# B&R Automation Studio project BenchEDM_AS6 (part 3)

#### TC_Recipe.fun - Exported functions and function blocks
```iecst
{REDUND_ERROR} FUNCTION_BLOCK TC_Recipe_Helper (*A helper block for MpRecipe*) (*$GROUP=User,$CAT=User,$GROUPICON=User.png,$CATICON=User.png*)
	VAR_INPUT
		Enable : BOOL;
		Def : Recipe_Definition_typ;
		RemOK : BOOL;
		ErrorReset : BOOL;
		ForceLoad : BOOL;
		ForceSave : BOOL;
		ForceDefaults : BOOL;
	END_VAR
	VAR_OUTPUT
		AutoLoadSuccess : BOOL;
		AutoLoadFailed : BOOL;
		RemLost : BOOL;
		Initialized : BOOL;
		Ready : BOOL;
		Error : BOOL;
	END_VAR
	VAR
		Internal : TC_Recipe_Helper_Internal_typ;
	END_VAR
END_FUNCTION_BLOCK
```

#### TC_Recipe_Helper.st
```iecst
(* A helper block for MpRecipe *)
FUNCTION_BLOCK TC_Recipe_Helper

//Reset in not enabled
	IF NOT Enable THEN
		Internal.State								:= TC_RH_ST_RESET;
	END_IF;

	//Reset Status Flags
	Ready 											:= FALSE;
	Error											:= FALSE;
	AutoLoadSuccess									:= FALSE;
	AutoLoadFailed									:= FALSE;
	RemLost											:= FALSE;

	//Main Case
	CASE Internal.State OF
		TC_RH_ST_RESET:
			Initialized								:= FALSE;
			Internal.ErrorReset 					:= FALSE;
			Internal.MpRecipeXml_0.Load				:= FALSE;
			Internal.MpRecipeXml_0.Save				:= FALSE;
			Internal.State							:= TC_RH_ST_VALIDATE_INPUTS;
		TC_RH_ST_VALIDATE_INPUTS:
			IF Def.pVar = 0 OR Def.SizeVar = 0 OR Def.DeviceName = '' OR Def.FileName = '' OR Def.VarName = '' THEN
				Internal.State						:= TC_RH_ST_ERROR;
			ELSE
				Internal.State						:= TC_RH_ST_REG_PAR_W;
			END_IF;
		TC_RH_ST_REG_PAR_W:
			Internal.CTON_Timeout.IN				:= TRUE;
			Internal.CTON_Timeout.PT				:= T#2s;
			IF Internal.MpRecipeRegPar_0.Error THEN
				Internal.State						:= TC_RH_ST_ERROR;
			ELSIF Internal.CTON_Timeout.Q THEN
				Internal.State						:= TC_RH_ST_ERROR;
			ELSIF Internal.MpRecipeRegPar_0.Active THEN
				IF RemOK THEN
					Internal.State					:= TC_RH_ST_READY;
				ELSE
					RemLost							:= TRUE;
					Internal.MpRecipeXml_0.Load		:= TRUE;
					Internal.State					:= TC_RH_ST_AUTO_LOAD_W;
				END_IF;
			END_IF;
		TC_RH_ST_READY:
			IF ForceLoad THEN
				Internal.MpRecipeXml_0.Load			:= TRUE;
				Internal.State						:= TC_RH_ST_LOAD_W;
			ELSIF ForceDefaults THEN
				IF Def.pDefaultVar <> 0 THEN
					brsmemcpy(Def.pVar,Def.pDefaultVar,Def.SizeVar);
				ELSE
					brsmemset(Def.pVar,0,Def.SizeVar);
				END_IF;
				Internal.MpRecipeXml_0.Save			:= TRUE;
				Internal.State						:= TC_RH_ST_SAVE_W;
			ELSIF ForceSave THEN
				Internal.MpRecipeXml_0.Save			:= TRUE;
				Internal.State						:= TC_RH_ST_SAVE_W;
			ELSIF Def.pCmpVar <> 0 THEN //AutoSave Enabled
				IF brsmemcmp(Def.pCmpVar,Def.pVar,Def.SizeVar) <> 0 THEN //AutoSave On Change
					brsmemcpy(Def.pCmpVar,Def.pVar,Def.SizeVar);
					Internal.MpRecipeXml_0.Save		:= TRUE;
					Internal.State					:= TC_RH_ST_SAVE_W;
				ELSE
					Ready 							:= TRUE;
					Initialized						:= TRUE;
				END_IF;
			ELSE
				Initialized							:= TRUE;
				Ready 								:= TRUE;
			END_IF;
		TC_RH_ST_LOAD_W:
			Internal.CTON_Timeout.IN				:= TRUE;
			Internal.CTON_Timeout.PT				:= T#2s;
			IF (NOT Internal.MpRecipeXml_0.CommandBusy AND Internal.MpRecipeXml_0.Error) OR Internal.CTON_Timeout.Q THEN
				Internal.MpRecipeXml_0.Load			:= FALSE;
				Internal.State						:= TC_RH_ST_ERROR;
			ELSIF (NOT Internal.MpRecipeXml_0.CommandBusy AND Internal.MpRecipeXml_0.CommandDone AND NOT Internal.MpRecipeXml_0.Error) THEN
				Internal.MpRecipeXml_0.Load			:= FALSE;
				Internal.State						:= TC_RH_ST_READY;
			END_IF;
		TC_RH_ST_SAVE_W:
			Internal.CTON_Timeout.IN				:= TRUE;
			Internal.CTON_Timeout.PT				:= T#2s;
			IF (NOT Internal.MpRecipeXml_0.CommandBusy AND Internal.MpRecipeXml_0.Error) OR Internal.CTON_Timeout.Q THEN
				Internal.MpRecipeXml_0.Save			:= FALSE;
				Internal.State						:= TC_RH_ST_ERROR;
			ELSIF (NOT Internal.MpRecipeXml_0.CommandBusy AND Internal.MpRecipeXml_0.CommandDone AND NOT Internal.MpRecipeXml_0.Error) THEN
				Internal.MpRecipeXml_0.Save			:= FALSE;
				Internal.State						:= TC_RH_ST_READY;
			END_IF;
		TC_RH_ST_AUTO_LOAD_W:
			Internal.CTON_Timeout.IN				:= TRUE;
			Internal.CTON_Timeout.PT				:= T#2s;
			IF (NOT Internal.MpRecipeXml_0.CommandBusy AND Internal.MpRecipeXml_0.Error) OR Internal.CTON_Timeout.Q THEN
				AutoLoadFailed						:= TRUE;
				IF Def.pDefaultVar <> 0 THEN
					brsmemcpy(Def.pVar,Def.pDefaultVar,Def.SizeVar);
				ELSE
					brsmemset(Def.pVar,0,Def.SizeVar);
				END_IF;
				Internal.MpRecipeXml_0.Load			:= FALSE;
				Internal.State						:= TC_RH_ST_AUTO_RESET_D;
			ELSIF (NOT Internal.MpRecipeXml_0.CommandBusy AND Internal.MpRecipeXml_0.CommandDone AND NOT Internal.MpRecipeXml_0.Error) THEN
				AutoLoadSuccess						:= TRUE;
				Internal.MpRecipeXml_0.Load			:= FALSE;
				Internal.State						:= TC_RH_ST_READY;
			END_IF;
		TC_RH_ST_AUTO_RESET_D:
			Internal.State							:= TC_RH_ST_AUTO_RESET_C;
		TC_RH_ST_AUTO_RESET_C:
			Internal.ErrorReset						:= TRUE;
			Internal.State							:= TC_RH_ST_AUTO_RESET_W;
		TC_RH_ST_AUTO_RESET_W:
			Internal.CTON_Timeout.IN				:= TRUE;
			Internal.CTON_Timeout.PT				:= T#2s;
			IF Internal.CTON_Timeout.Q THEN
				Internal.ErrorReset					:= FALSE;
				Internal.State						:= TC_RH_ST_ERROR;
			ELSIF NOT Internal.MpRecipeXml_0.Error THEN
				Internal.ErrorReset					:= FALSE;
				Internal.MpRecipeXml_0.Save			:= TRUE;
				Internal.State						:= TC_RH_ST_AUTO_SAVE_W;
			END_IF;
		TC_RH_ST_AUTO_SAVE_W:
			Internal.CTON_Timeout.IN				:= TRUE;
			Internal.CTON_Timeout.PT				:= T#2s;
			IF (NOT Internal.MpRecipeXml_0.CommandBusy AND Internal.MpRecipeXml_0.Error) OR Internal.CTON_Timeout.Q THEN
				Internal.MpRecipeXml_0.Save			:= FALSE;
				Internal.State						:= TC_RH_ST_ERROR;
			ELSIF (NOT Internal.MpRecipeXml_0.CommandBusy AND Internal.MpRecipeXml_0.CommandDone AND NOT Internal.MpRecipeXml_0.Error) THEN
				Internal.MpRecipeXml_0.Save			:= FALSE;
				Internal.State						:= TC_RH_ST_READY;
			END_IF;
		TC_RH_ST_ERROR:
			Error									:= TRUE;
			IF ErrorReset THEN
				Internal.State						:= TC_RH_ST_RESET;
			END_IF;
	END_CASE;

	//Reset Commands
	ForceDefaults 									:= FALSE;
	ForceLoad 										:= FALSE;
	ForceSave 										:= FALSE;

	//Reset Timeout On State Change
	IF Internal.LastState <> Internal.State OR Internal.State = TC_RH_ST_RESET THEN
		Internal.LastState 							:= Internal.State;
		Internal.CTON_Timeout.IN					:= FALSE;
	END_IF;

	//FB Calls
	Internal.CTON_Timeout();
	Internal.MpRecipeRegPar_0(MpLink := ADR(Def.MpLink), Enable := Enable, ErrorReset := (ErrorReset OR Internal.ErrorReset), PVName := ADR(Def.VarName), Category := ADR(Def.VarName));
	Internal.MpRecipeXml_0(MpLink := ADR(Def.MpLink), Enable := Enable, ErrorReset := (ErrorReset OR Internal.ErrorReset), DeviceName := ADR(Def.DeviceName), FileName := ADR(Def.FileName), Category := ADR(Def.VarName));

END_FUNCTION_BLOCK
```

### Library Logical/Libraries/TC_Sim (IEC)
Depends on: MTTypes, MTBasics, MTFilter

#### Types.typ - Exported data types
```iecst
TYPE
	TC_Sim_Actuator_TF_Internal_typ : 	STRUCT
		Active : BOOL;
		OldDampingRatio : REAL;
		OldNaturalFreq : REAL;
		OldFullStrokeValue : REAL;
		MTBasicsTransferFcn_0 : MTBasicsTransferFcn;
	END_STRUCT;
	TC_Sim_Actuator_Lin_Internal_typ : 	STRUCT
		Active : BOOL;
		OldTimePos : REAL;
		OldTimeNeg : REAL;
		MTBasicsLimiter_0 : MTBasicsLimiter;
	END_STRUCT;
END_TYPE
```

#### TC_Sim.fun - Exported functions and function blocks
```iecst
{REDUND_ERROR} FUNCTION_BLOCK TC_Sim_Actuator_Lin (* *) (*$GROUP=User,$CAT=User,$GROUPICON=User.png,$CATICON=User.png*)
	VAR_INPUT
		Enable : BOOL;
		Actuate : BOOL;
		FullStrokeValue : REAL;
		FeedbackTol : REAL;
		TimeNeg : REAL;
		TimePos : REAL;
	END_VAR
	VAR_OUTPUT
		Position : REAL;
		AtFalsePosition : BOOL;
		AtTruePosition : BOOL;
		Error : BOOL;
	END_VAR
	VAR
		Internal : TC_Sim_Actuator_Lin_Internal_typ;
	END_VAR
END_FUNCTION_BLOCK

{REDUND_ERROR} FUNCTION_BLOCK TC_Sim_Actuator_TF (* *) (*$GROUP=User,$CAT=User,$GROUPICON=User.png,$CATICON=User.png*)
	VAR_INPUT
		Enable : BOOL;
		Actuate : BOOL;
		ClampValueToEnds : BOOL;
		FullStrokeValue : REAL;
		FeedbackTol : REAL;
		NaturalFreq : REAL;
		DampingRatio : REAL;
	END_VAR
	VAR_OUTPUT
		Position : REAL;
		AtFalsePosition : BOOL;
		AtTruePosition : BOOL;
		Error : BOOL;
	END_VAR
	VAR
		Internal : TC_Sim_Actuator_TF_Internal_typ;
	END_VAR
END_FUNCTION_BLOCK
```

#### TC_Sim_Actuator_TF.st
```iecst
FUNCTION_BLOCK TC_Sim_Actuator_TF

	IF Enable THEN
		IF NOT Internal.Active OR (Internal.Active AND (Internal.OldNaturalFreq <> NaturalFreq OR Internal.OldDampingRatio <> DampingRatio OR Internal.OldFullStrokeValue <> FullStrokeValue)) THEN
			Internal.MTBasicsTransferFcn_0.Numerator[0] 	:= FullStrokeValue*NaturalFreq**2;
			Internal.MTBasicsTransferFcn_0.Denominator[0] 	:= NaturalFreq**2;
			Internal.MTBasicsTransferFcn_0.Denominator[1] 	:= 2*DampingRatio*NaturalFreq;
			Internal.MTBasicsTransferFcn_0.Denominator[2] 	:= 1;
			Internal.OldNaturalFreq							:= NaturalFreq;
			Internal.OldDampingRatio						:= DampingRatio;
			Internal.OldFullStrokeValue						:= FullStrokeValue;
			IF Internal.Active THEN
				Internal.MTBasicsTransferFcn_0.Update		:= TRUE;
			END_IF;
			Internal.Active 								:= TRUE;
		END_IF;

		IF Actuate THEN
			Internal.MTBasicsTransferFcn_0.In				:= 1.0;
		ELSE
			Internal.MTBasicsTransferFcn_0.In				:= 0.0;
		END_IF;

		Position 											:= Internal.MTBasicsTransferFcn_0.Out;
		IF ClampValueToEnds THEN
			IF Internal.MTBasicsTransferFcn_0.Out > FullStrokeValue THEN
				Position 									:= FullStrokeValue;
			ELSIF Internal.MTBasicsTransferFcn_0.Out < 0 THEN
				Position 									:= 0.0;
			END_IF;
		END_IF;

		AtFalsePosition										:= ABS(Position) <= FeedbackTol;
		AtTruePosition										:= ABS(Position-FullStrokeValue) <= FeedbackTol;
		Internal.MTBasicsTransferFcn_0.Enable				:= TRUE;
	ELSE
		Position 											:= 0.0;
		AtFalsePosition 									:= FALSE;
		AtTruePosition 										:= FALSE;
		Internal.Active 									:= FALSE;
		Internal.MTBasicsTransferFcn_0.Enable				:= FALSE;
		Internal.MTBasicsTransferFcn_0.In					:= 0.0;
		Internal.OldNaturalFreq								:= 0.0;
		Internal.OldDampingRatio							:= 0.0;
		Internal.OldFullStrokeValue							:= 0.0;
	END_IF;

	Internal.MTBasicsTransferFcn_0();
	Internal.MTBasicsTransferFcn_0.Update 					:= FALSE;
	Error 													:= Internal.MTBasicsTransferFcn_0.Error;

END_FUNCTION_BLOCK
```

#### TC_Sim_Actuator_Lin.st
```iecst
FUNCTION_BLOCK TC_Sim_Actuator_Lin

	IF Enable THEN
		IF NOT Internal.Active OR (Internal.Active AND (Internal.OldTimeNeg <> TimeNeg OR Internal.OldTimePos <> TimePos)) THEN
			IF TimeNeg <= 0 THEN
				Internal.MTBasicsLimiter_0.MaxNegSlewRate	:= 0;
			ELSE
				Internal.MTBasicsLimiter_0.MaxNegSlewRate	:= 1.0/TimeNeg;
			END_IF;
			IF TimePos <= 0 THEN
				Internal.MTBasicsLimiter_0.MaxPosSlewRate	:= 0;
			ELSE
				Internal.MTBasicsLimiter_0.MaxPosSlewRate	:= 1.0/TimePos;
			END_IF;
			Internal.OldTimeNeg 							:= TimeNeg;
			Internal.OldTimePos 							:= TimePos;
			IF Internal.Active THEN
				Internal.MTBasicsLimiter_0.Update			:= TRUE;
			END_IF;
			Internal.Active 								:= TRUE;
		END_IF;

		IF Actuate THEN
			Internal.MTBasicsLimiter_0.In					:= 1.0;
		ELSE
			Internal.MTBasicsLimiter_0.In					:= 0.0;
		END_IF;

		Position 											:= Internal.MTBasicsLimiter_0.Out*FullStrokeValue;

		AtFalsePosition										:= ABS(Position) <= FeedbackTol;
		AtTruePosition										:= ABS(Position-FullStrokeValue) <= FeedbackTol;
		Internal.MTBasicsLimiter_0.Enable					:= TRUE;
	ELSE
		Position 											:= 0.0;
		AtFalsePosition 									:= FALSE;
		AtTruePosition 										:= FALSE;
		Internal.Active 									:= FALSE;
		Internal.MTBasicsLimiter_0.Enable					:= FALSE;
		Internal.MTBasicsLimiter_0.In						:= 0.0;
		Internal.OldTimeNeg									:= 0.0;
		Internal.OldTimePos									:= 0.0;
	END_IF;

	Internal.MTBasicsLimiter_0();
	Internal.MTBasicsLimiter_0.Update 						:= FALSE;
	Error 													:= Internal.MTBasicsLimiter_0.Error;

END_FUNCTION_BLOCK
```

### Library Logical/Libraries/TC_AlarmX (IEC)
Depends on: AsBrStr, TC_General, TC_Str, MpAlarmX, MpBase

#### Types.typ - Exported data types
```iecst
TYPE
	TC_AlarmX_Helper_Internal_typ : 	STRUCT
		Active : BOOL;
		AddText : STRING[1000];
		ArEventLogGetIdent_0 : ArEventLogGetIdent;
		ArEventLogWrite_0 : ArEventLogWrite;
	END_STRUCT;
	TC_ALARMX_ACTION_ENUM :
		(
		TC_ALARMX_ACTION_NONE,
		TC_ALARMX_ACTION_SET,
		TC_ALARMX_ACTION_SET_NO_LOG,
		TC_ALARMX_ACTION_ACK,
		TC_ALARMX_ACTION_ACK_NO_LOG,
		TC_ALARMX_ACTION_LOG_ONLY
		);
	TC_ALARMX_CORE_STATE_ENUM :
		(
		TC_ALARMX_CORE_RESET,
		TC_ALARMX_CORE_IDLE,
		TC_ALARMX_CORE_SET_C,
		TC_ALARMX_CORE_SET_W
		);
	TC_AlarmX_Core_Internal_typ : 	STRUCT
		state : TC_ALARMX_CORE_STATE_ENUM;
		currentAlarm : TC_AlarmX_Core_Buffer_typ;
		tDelay : CTON;
		i : INT;
	END_STRUCT;
	TC_AlarmX_Core_Buffer_typ : 	STRUCT
		name : STRING[MAX_ALARM_NAME_LEN];
		addText : ARRAY[0..TC_ALARMX_MAX_ADD_DATA_IDX]OF STRING[MAX_ALARM_ADD_DATA];
		allowMultiple : BOOL;
	END_STRUCT;
	TC_AlarmX_AlarmExtraData_typ : 	STRUCT
		AddData : ARRAY[0..TC_ALARMX_MAX_ADD_DATA_IDX]OF STRING[MAX_ALARM_ADD_DATA];
	END_STRUCT;
	TC_AlarmX_CfgMod_Internal_typ : 	STRUCT
		AlarmName : STRING[MAX_ALARM_NAME_LEN];
		i : USINT;
		CTON_Timeout : CTON;
	END_STRUCT;
	TC_AlarmX_BufferInfo_typ : 	STRUCT
		Address : UDINT;
		Size : UDINT;
	END_STRUCT;
	TC_Module_Alarm_Info_typ : 	STRUCT
		ErrorInfo : USINT;
		IgnoreInfo : USINT;
	END_STRUCT;
END_TYPE
```

#### Constants.var - Exported constants
```iecst
VAR CONSTANT
	TC_MODULE_MAX_ALARM : USINT := 6;
	MAX_ALARM_ADD_DATA : UDINT := 255; (*Maximum Length of the extra alarm text*)
	MAX_ALARM_NAME_LEN : UDINT := 255; (*Maximum Length of the alarm name*)
	TC_ALARMX_BUFFER_IDX : UDINT := 255; (*Length of alarm buffer*)
	TC_ALARMX_MAX_ADD_DATA_IDX : USINT := 3;
END_VAR
```

#### TC_AlarmX.fun - Exported functions and function blocks
```iecst
{REDUND_ERROR} FUNCTION TC_AlarmX_Helper : DINT (*Helper Function for Setting and Acknowledging Alarms with User Logger support.*) (*$GROUP=User,$CAT=User,$GROUPICON=User.png,$CATICON=User.png*)
	VAR_INPUT
		MpLink : MpComIdentType;
		AlarmName : STRING[255];
		AlarmAction : TC_ALARMX_ACTION_ENUM;
		LogEventAddText : STRING[255];
		AllowMultiple : BOOL;
	END_VAR
	VAR
		Internal : TC_AlarmX_Helper_Internal_typ;
	END_VAR
END_FUNCTION

{REDUND_ERROR} FUNCTION_BLOCK TC_AlarmXCore (*TODO: Add your comment here*) (*$GROUP=User,$CAT=User,$GROUPICON=User.png,$CATICON=User.png*)
	VAR_INPUT
		enable : BOOL;
		MpLink : MpComIdentType;
		pBuffer : UDINT;
		pOutputData : REFERENCE TO TC_AlarmX_AlarmExtraData_typ;
		delayTime : TIME;
	END_VAR
	VAR
		internal : TC_AlarmX_Core_Internal_typ;
	END_VAR
END_FUNCTION_BLOCK
```

#### TC_AlarmX_Helper.st
```iecst
(* Helper Function for Setting and Acknowledging Alarms with User Logger support. *)
FUNCTION TC_AlarmX_Helper
	TC_AlarmX_Helper 					:= -1;
	brsmemset(ADR(Internal),0,SIZEOF(Internal));
	Internal.ArEventLogGetIdent_0(Execute := FALSE);
	Internal.ArEventLogGetIdent_0(Execute := TRUE, Name := '$$arlogusr');
	Internal.AddText 					:= AlarmName;
	Internal.Active						:= NOT MpAlarmXCheckState(MpLink,AlarmName,mpALARMX_STATE_NONE);

	CASE AlarmAction OF
		TC_ALARMX_ACTION_NONE:
			TC_AlarmX_Helper 			:= 0;
		TC_ALARMX_ACTION_SET:
			TC_AlarmX_Helper 			:= 0;
			IF NOT Internal.Active OR AllowMultiple THEN
				MpAlarmXSet(MpLink,AlarmName);
				brsmemset(ADR(Internal.AddText),0,SIZEOF(Internal.AddText));
				Internal.AddText 	:= AlarmName;
				TC_brsstrcat(ADR(Internal.AddText),ADR(' - Set'),SIZEOF(Internal.AddText));
				IF LogEventAddText <> '' THEN
					TC_brsstrcat(ADR(Internal.AddText),ADR(' - Info: '),SIZEOF(Internal.AddText));
					TC_brsstrcat(ADR(Internal.AddText),ADR(LogEventAddText),SIZEOF(Internal.AddText));
				END_IF;
				Internal.ArEventLogWrite_0(Execute := FALSE);
				Internal.ArEventLogWrite_0(Execute := TRUE, Ident := Internal.ArEventLogGetIdent_0.Ident, EventID := -536870912, OriginRecordID := 0, ObjectID := 'TC_AlarmX_Helper', AddDataSize := brsstrlen(ADR(Internal.AddText)), AddDataFormat := 1, AddData := ADR(Internal.AddText), TimeStamp := 0);
			END_IF;
		TC_ALARMX_ACTION_SET_NO_LOG:
			TC_AlarmX_Helper 			:= 0;
			IF NOT Internal.Active OR AllowMultiple THEN
				MpAlarmXSet(MpLink,AlarmName);
				brsmemset(ADR(Internal.AddText),0,SIZEOF(Internal.AddText));
			END_IF;
		TC_ALARMX_ACTION_ACK:
			TC_AlarmX_Helper 			:= 0;
			IF Internal.Active THEN
				MpAlarmXAcknowledge(MpLink,AlarmName);
				brsmemset(ADR(Internal.AddText),0,SIZEOF(Internal.AddText));
				Internal.AddText 	:= AlarmName;
				TC_brsstrcat(ADR(Internal.AddText),ADR(' - Ack'),SIZEOF(Internal.AddText));
				IF LogEventAddText <> '' THEN
					TC_brsstrcat(ADR(Internal.AddText),ADR(' - Info: '),SIZEOF(Internal.AddText));
					TC_brsstrcat(ADR(Internal.AddText),ADR(LogEventAddText),SIZEOF(Internal.AddText));
				END_IF;
				Internal.ArEventLogWrite_0(Execute := FALSE);
				Internal.ArEventLogWrite_0(Execute := TRUE, Ident := Internal.ArEventLogGetIdent_0.Ident, EventID := -536870912, OriginRecordID := 0, ObjectID := 'TC_AlarmX_Helper', AddDataSize := brsstrlen(ADR(Internal.AddText)), AddDataFormat := 1, AddData := ADR(Internal.AddText), TimeStamp := 0);
			END_IF;
		TC_ALARMX_ACTION_ACK_NO_LOG:
			TC_AlarmX_Helper 			:= 0;
			IF Internal.Active THEN
				MpAlarmXAcknowledge(MpLink,AlarmName);
			END_IF;
		TC_ALARMX_ACTION_LOG_ONLY:
			TC_AlarmX_Helper 			:= 0;
			brsmemset(ADR(Internal.AddText),0,SIZEOF(Internal.AddText));
			IF LogEventAddText <> '' THEN
				TC_brsstrcat(ADR(Internal.AddText),ADR('Info: '),SIZEOF(Internal.AddText));
				TC_brsstrcat(ADR(Internal.AddText),ADR(LogEventAddText),SIZEOF(Internal.AddText));
				Internal.ArEventLogWrite_0(Execute := FALSE);
				Internal.ArEventLogWrite_0(Execute := TRUE, Ident := Internal.ArEventLogGetIdent_0.Ident, EventID := -536870912, OriginRecordID := 0, ObjectID := 'TC_AlarmX_Helper', AddDataSize := brsstrlen(ADR(Internal.AddText)), AddDataFormat := 1, AddData := ADR(Internal.AddText), TimeStamp := 0);
			END_IF;
	END_CASE;

END_FUNCTION
```

#### TC_AlarmXCore.st
```iecst
(* Alarm Core to handle setting multiple alarms in one cycle with different texts *)
FUNCTION_BLOCK TC_AlarmXCore

	IF enable = FALSE THEN
		internal.state := TC_ALARMX_CORE_RESET;
	END_IF

	CASE internal.state OF

		TC_ALARMX_CORE_RESET:

			brsmemset(ADR(internal.currentAlarm), 0, SIZEOF(internal.currentAlarm));
			internal.state := TC_ALARMX_CORE_IDLE;

		TC_ALARMX_CORE_IDLE:

			IF TC_Array_PeekBtm(pBuffer, SIZEOF(internal.currentAlarm) * TC_ALARMX_BUFFER_IDX, ADR(internal.currentAlarm), SIZEOF(internal.currentAlarm)) > 0 THEN
				TC_Array_Dequeue(pBuffer, SIZEOF(internal.currentAlarm) * TC_ALARMX_BUFFER_IDX, ADR(internal.currentAlarm), SIZEOF(internal.currentAlarm));
				internal.state := TC_ALARMX_CORE_SET_C;
			END_IF

		TC_ALARMX_CORE_SET_C:

			FOR internal.i := 0 TO TC_ALARMX_MAX_ADD_DATA_IDX DO
				pOutputData.AddData[internal.i]	:= internal.currentAlarm.addText[internal.i];
			END_FOR
			TC_AlarmX_Helper(MpLink, internal.currentAlarm.name, TC_ALARMX_ACTION_SET, '', internal.currentAlarm.allowMultiple);

			internal.state := TC_ALARMX_CORE_SET_W;

		TC_ALARMX_CORE_SET_W:

			internal.tDelay.IN	:= TRUE;
			internal.tDelay.PT	:= delayTime;

			IF internal.tDelay.Q THEN
				internal.tDelay.IN	:= FALSE;
				internal.state 		:= TC_ALARMX_CORE_IDLE;
			END_IF

	END_CASE

	internal.tDelay();

END_FUNCTION_BLOCK
```

### Library Logical/Libraries/TC_Str (IEC)

#### Types.typ - Exported data types
```iecst
TYPE
	TC_brsstrcat_Internal_typ : 	STRUCT
		SrcSize : UDINT;
		DestSize : UDINT;
	END_STRUCT;
	TC_Find_Extract_Internal_typ : 	STRUCT
		i : UDINT;
		sB : UDINT;
		sSL : UDINT;
		sSR : UDINT;
		Len : UDINT;
		Pos : UDINT;
		P1 : DINT;
		P2 : DINT;
	END_STRUCT;
	TC_Find_S_Internal_typ : 	STRUCT
		i : UDINT;
		sB : UDINT;
		sS : UDINT;
	END_STRUCT;
	TC_Find_R_Internal_typ : 	STRUCT
		i : UDINT;
		sB : UDINT;
		sS : UDINT;
	END_STRUCT;
	TC_Find_L_Internal_typ : 	STRUCT
		i : UDINT;
		sB : UDINT;
		sS : UDINT;
	END_STRUCT;
END_TYPE
```

#### TC_Str.fun - Exported functions and function blocks
```iecst
FUNCTION TC_brsstrcat : BOOL
	VAR_INPUT
		pDest : UDINT;
		pSrc : UDINT;
		DestSize : UDINT;
	END_VAR
	VAR
		Internal : TC_brsstrcat_Internal_typ;
	END_VAR
END_FUNCTION

{REDUND_ERROR} FUNCTION TC_Find_L : DINT (*Returns index of substring. Negative values are Errors.*) (*$GROUP=User,$CAT=User,$GROUPICON=User.png,$CATICON=User.png*)
	VAR_INPUT
		pBuffer : UDINT;
		pSearch : UDINT;
	END_VAR
	VAR
		Internal : TC_Find_L_Internal_typ;
	END_VAR
END_FUNCTION

{REDUND_ERROR} FUNCTION TC_Find_R : DINT (*Returns right index of substring. Negative values are Errors.*) (*$GROUP=User,$CAT=User,$GROUPICON=User.png,$CATICON=User.png*)
	VAR_INPUT
		pBuffer : UDINT;
		pSearch : UDINT;
	END_VAR
	VAR
		Internal : TC_Find_R_Internal_typ;
	END_VAR
END_FUNCTION

{REDUND_ERROR} FUNCTION TC_Find_S : DINT (*Returns right index of substring. Negative values are Errors.*) (*$GROUP=User,$CAT=User,$GROUPICON=User.png,$CATICON=User.png*)
	VAR_INPUT
		pBuffer : UDINT;
		pSearch : UDINT;
	END_VAR
	VAR
		Internal : TC_Find_S_Internal_typ;
	END_VAR
END_FUNCTION

{REDUND_ERROR} FUNCTION TC_Find_Extract : DINT (*Returns end position for next search. Negative values are Errors.*) (*$GROUP=User,$CAT=User,$GROUPICON=User.png,$CATICON=User.png*)
	VAR_INPUT
		pBuffer : UDINT;
		pSearchL : UDINT;
		pSearchR : UDINT;
		pExtractADR : UDINT;
		pExtractSIZEOF : UDINT;
	END_VAR
	VAR
		Internal : TC_Find_Extract_Internal_typ;
	END_VAR
END_FUNCTION
```

#### TC_brsstrcat.st
```iecst
(* Checks the memory area before concatenating to prevent overrun. Returns false and doesnt concat if overrun is detected *)
FUNCTION TC_brsstrcat
	TC_brsstrcat 						:= TRUE;
	IF pSrc = 0 OR pDest = 0 OR DestSize = 0 THEN
		TC_brsstrcat 					:= FALSE;
	ELSE
		TC_brsstrcat					:= TRUE;
		brsmemset(ADR(Internal),0,SIZEOF(Internal));
		Internal.SrcSize := brsstrlen(pSrc);
		Internal.DestSize := brsstrlen(pDest);
		IF (Internal.SrcSize+Internal.DestSize) <= DestSize-1 THEN
			brsstrcat(pDest,pSrc);
		ELSE
			TC_brsstrcat				:= FALSE;
		END_IF;
	END_IF;
END_FUNCTION
```

#### TC_Find_S.st
```iecst
(* Returns Right index of substring, substring only returns result if found at START of buffer. Negative values are Errors. *)
FUNCTION TC_Find_S
	IF pBuffer = 0 OR pSearch = 0 THEN
		TC_Find_S	 						:= -2;
	ELSE
		Internal.sB							:= brsstrlen(pBuffer);
		Internal.sS							:= brsstrlen(pSearch);
		IF Internal.sB = 0 OR Internal.sB < Internal.sS THEN
		TC_Find_S	 						:= -3;
		END_IF;
	END_IF;
	IF TC_Find_S = 0 THEN
		TC_Find_S							:= -1;
		IF Internal.sS = 0 THEN
			TC_Find_S 						:= 0;
			RETURN;
		ELSE
			FOR Internal.i := 0 TO Internal.sB-Internal.sS DO
				IF brsmemcmp(pBuffer+Internal.i,pSearch,Internal.sS) = 0 THEN
					TC_Find_S 				:= Internal.i+Internal.sS;
					RETURN;
				ELSE
					RETURN;
				END_IF;
			END_FOR;
		END_IF;
	END_IF;
END_FUNCTION
```

#### TC_Find_L.st
```iecst
(* Returns Left index of substring. Negative values are Errors. *)
FUNCTION TC_Find_L
	IF pBuffer = 0 OR pSearch = 0 THEN
		TC_Find_L	 						:= -2;
	ELSE
		Internal.sB							:= brsstrlen(pBuffer);
		Internal.sS							:= brsstrlen(pSearch);
		IF Internal.sB = 0 OR Internal.sB < Internal.sS THEN
			TC_Find_L	 					:= -3;
		END_IF;
	END_IF;
	IF TC_Find_L = 0 THEN
		TC_Find_L							:= -1;
		IF Internal.sS = 0 THEN
			TC_Find_L 						:= 0;
			RETURN;
		ELSE
			FOR Internal.i := 0 TO Internal.sB-Internal.sS DO
				IF brsmemcmp(pBuffer+Internal.i,pSearch,Internal.sS) = 0 THEN
					TC_Find_L 				:= Internal.i;
					RETURN;
				END_IF;
			END_FOR;
		END_IF;
	END_IF;
END_FUNCTION
```

#### TC_Find_R.st
```iecst
(* Returns Right index of substring. Negative values are Errors. *)
FUNCTION TC_Find_R
	IF pBuffer = 0 OR pSearch = 0 THEN
		TC_Find_R	 						:= -2;
	ELSE
		Internal.sB							:= brsstrlen(pBuffer);
		Internal.sS							:= brsstrlen(pSearch);
		IF Internal.sB = 0 OR Internal.sB < Internal.sS THEN
		TC_Find_R	 						:= -3;
		END_IF;
	END_IF;
	IF TC_Find_R = 0 THEN
		TC_Find_R							:= -1;
		IF Internal.sS = 0 THEN
			TC_Find_R 						:= 0;
			RETURN;
		ELSE
			FOR Internal.i := 0 TO Internal.sB-Internal.sS DO
				IF brsmemcmp(pBuffer+Internal.i,pSearch,Internal.sS) = 0 THEN
					TC_Find_R 				:= Internal.i+Internal.sS;
					RETURN;
				END_IF;
			END_FOR;
		END_IF;
	END_IF;
END_FUNCTION
```

#### TC_Find_Extract.st
```iecst
(* Negative values are Errors. *)
FUNCTION TC_Find_Extract
	IF pBuffer = 0 OR pSearchL = 0 OR pSearchR = 0 OR pExtractADR = 0 OR pExtractSIZEOF = 0 THEN
		TC_Find_Extract 						:= -2;
	ELSE
		Internal.sB								:= brsstrlen(pBuffer);
		Internal.sSL							:= brsstrlen(pSearchL);
		Internal.sSR							:= brsstrlen(pSearchR);
		IF Internal.sB = 0 OR Internal.sB < (Internal.sSL + Internal.sSR + 1) THEN
			TC_Find_Extract 					:= -3;
		END_IF;
	END_IF;
	IF TC_Find_Extract = 0 THEN
		TC_Find_Extract							:= -1;
		Internal.P1 							:= TC_Find_R(pBuffer,pSearchL);
		IF Internal.P1 >= 0 THEN
			Internal.P2 						:= TC_Find_L(pBuffer+Internal.P1,pSearchR);
			IF Internal.P2 >= 0 THEN
				Internal.Pos 					:= Internal.P1 + pBuffer;
				Internal.Len 					:= DINT_TO_UDINT(Internal.P2);
				brsmemcpy(pExtractADR,ADR(Internal.Pos),4);
				brsmemcpy(pExtractSIZEOF,ADR(Internal.Len),4);
				TC_Find_Extract					:= Internal.P1+Internal.P2+Internal.sSR;
			END_IF;
		END_IF;
	END_IF;
END_FUNCTION
```

### Library Logical/Libraries/TC_JSON (IEC)
Depends on: TC_Str, AsBrStr, sys_lib

#### TC_JSON.fun - Exported functions and function blocks
```iecst
{REDUND_ERROR} FUNCTION_BLOCK TC_JSON_PairsToJSON (*FB parses a JSON string into a flat array of Name and Value Pairs*) (*$GROUP=User,$CAT=User,$GROUPICON=User.png,$CATICON=User.png*)
	VAR_INPUT
		Enable : BOOL;
		pBuffer : UDINT; (*Pointer to Buffer*)
		BufferSIZEOF : UDINT; (*Buffer SIZEOF*)
		pPairs : UDINT; (*Pointer to Array defined as HA_JSON_Parse_Pair_typ[0..MAX_JSON_PARSE_PAIR_IDX]*)
	END_VAR
	VAR_OUTPUT
		Done : BOOL;
		Error : BOOL;
	END_VAR
	VAR
		Internal : TC_JSON_PairsToJSON_Internal_typ;
	END_VAR
END_FUNCTION_BLOCK

{REDUND_ERROR} FUNCTION_BLOCK TC_JSON_Parse (*FB parses a JSON string into a flat array of Name and Value Pairs*) (*$GROUP=User,$CAT=User,$GROUPICON=User.png,$CATICON=User.png*)
	VAR_INPUT
		Enable : BOOL;
		pBuffer : UDINT; (*Pointer to Buffer*)
		pPairs : UDINT; (*Pointer to Array defined as TC_JSON_Parse_Pair_typ[0..MAX_JSON_PARSE_PAIR_IDX]*)
		NoQuotes : BOOL; (*Pointer to Array defined as HA_JSON_Parse_Pair_typ[0..MAX_JSON_PARSE_PAIR_IDX]*)
	END_VAR
	VAR_OUTPUT
		Done : BOOL;
		Error : BOOL;
	END_VAR
	VAR
		Internal : TC_JSON_Parse_Internal_typ;
	END_VAR
END_FUNCTION_BLOCK
```

#### Types.typ - Exported data types
```iecst
TYPE
	TC_JSON_PairsToJSON_Internal_typ : 	STRUCT
		Depth : DINT;
		DepthArrayIdx : ARRAY[0..MAX_JSON_PARSE_DEPTH_IDX]OF DINT;
		Enabled : BOOL;
		j : DINT;
		i : DINT;
		Pair : TC_JSON_Parse_Pair_typ;
	END_STRUCT;
	TC_JSON_Parse_Internal_typ : 	STRUCT
		Depth : DINT;
		DepthArrayIdx : ARRAY[0..MAX_JSON_PARSE_DEPTH_IDX]OF DINT;
		DepthIDs : ARRAY[0..MAX_JSON_PARSE_DEPTH_IDX]OF STRING[MAX_JSON_PARSE_NAME_LEN];
		Marker : UDINT;
		InValueNonWhiteFound : BOOL;
		InValue : BOOL;
		InQuote : BOOL;
		QuoteIsDouble : BOOL;
		Send : BOOL;
		Idx : DINT;
		i : DINT;
		Enabled : BOOL;
		BufferLEN : UDINT;
		Pair : TC_JSON_Parse_Pair_typ;
	END_STRUCT;
	TC_JSON_Parse_Pair_typ : 	STRUCT
		Name : STRING[MAX_JSON_PARSE_NAME_LEN];
		Value : STRING[MAX_JSON_PARSE_VALUE_LEN];
	END_STRUCT;
END_TYPE
```

#### Constants.var - Exported constants
```iecst
VAR CONSTANT
	MAX_JSON_PARSE_DEPTH_IDX : DINT := 4;
	MAX_JSON_PARSE_PAIR_IDX : DINT := 19;
	MAX_JSON_PARSE_NAME_LEN : DINT := 40;
	MAX_JSON_PARSE_VALUE_LEN : DINT := 255;
END_VAR
```

#### TC_JSON_Parse.st
```iecst
(* FB parses a JSON string into a flat array of Name and Value Pairs, FOR LOOP COMPATIBLE *)FUNCTION_BLOCK TC_JSON_Parse

	IF Enable THEN
		IF NOT Internal.Enabled THEN
			brsmemset(ADR(Internal),0,SIZEOF(Internal));
			brsmemset(pPairs,0,(SIZEOF(Internal.Pair)*(MAX_JSON_PARSE_PAIR_IDX+1)));
			Internal.BufferLEN												:= brsstrlen(pBuffer);
			Internal.DepthArrayIdx[0]										:= -1;
			Internal.Enabled												:= TRUE;
		END_IF;
		IF Error OR Done THEN
			// Do Nothing, Enable must be toggled to parse again
		ELSE
			FOR Internal.i := 0 TO UDINT_TO_DINT(Internal.BufferLEN) DO
				IF NOT Internal.InQuote THEN
					IF TC_Find_S(pBuffer+Internal.i,ADR('[')) >= 0 THEN													// New Array
						IF Internal.Depth <= MAX_JSON_PARSE_DEPTH_IDX THEN
							Internal.Depth 									:= Internal.Depth + 1;
							Internal.DepthIDs[Internal.Depth]				:= Internal.Pair.Name;
							IF Internal.DepthArrayIdx[Internal.Depth-1] >= 0 THEN
								Internal.Pair.Name							:= DINT_TO_STRING(Internal.DepthArrayIdx[Internal.Depth-1]);
								Internal.DepthArrayIdx[Internal.Depth-1] := Internal.DepthArrayIdx[Internal.Depth-1] + 1;
							END_IF;
							Internal.Pair.Value								:= '[';
							Internal.DepthIDs[Internal.Depth]				:= Internal.Pair.Name;
							Internal.DepthArrayIdx[Internal.Depth]			:= 0;
							Internal.Send									:= TRUE;
						ELSE
							Error											:= TRUE;
							EXIT;
						END_IF;
					ELSIF TC_Find_S(pBuffer+Internal.i,ADR('{')) >= 0 THEN 												// New Struct
						IF Internal.Depth <= MAX_JSON_PARSE_DEPTH_IDX THEN
							Internal.Depth 									:= Internal.Depth + 1;
							IF Internal.DepthArrayIdx[Internal.Depth-1] >= 0 THEN
								Internal.Pair.Name							:= DINT_TO_STRING(Internal.DepthArrayIdx[Internal.Depth-1]);
								Internal.DepthIDs[Internal.Depth]			:= Internal.Pair.Name;
								Internal.DepthArrayIdx[Internal.Depth-1] 	:= Internal.DepthArrayIdx[Internal.Depth-1] + 1;
								Internal.DepthArrayIdx[Internal.Depth]		:= -1;
								Internal.Pair.Value							:= '{';
								Internal.Send								:= TRUE;
							ELSE
								Internal.DepthIDs[Internal.Depth]			:= Internal.Pair.Name;
								Internal.DepthArrayIdx[Internal.Depth]		:= -1;
								Internal.Pair.Value							:= '{';
								Internal.Send								:= TRUE;
							END_IF;
						ELSE
							Error											:= TRUE;
							EXIT;
						END_IF;
					ELSIF TC_Find_S(pBuffer+Internal.i,ADR('"')) >= 0 THEN 												// New Double Quote
						Internal.InQuote									:= TRUE;
						Internal.QuoteIsDouble								:= TRUE;
						Internal.Marker										:= Internal.i+1;
						IF Internal.DepthArrayIdx[Internal.Depth] >= 0 THEN
							Internal.Pair.Name								:= DINT_TO_STRING(Internal.DepthArrayIdx[Internal.Depth]);
							Internal.DepthArrayIdx[Internal.Depth] 			:= Internal.DepthArrayIdx[Internal.Depth] + 1;
							Internal.InValue								:= TRUE;
						END_IF;
					ELSIF TC_Find_S(pBuffer+Internal.i,ADR('$'')) >= 0 THEN 											// New Single Quote
						Internal.InQuote									:= TRUE;
						Internal.QuoteIsDouble								:= FALSE;
						Internal.Marker										:= Internal.i+1;
						IF Internal.DepthArrayIdx[Internal.Depth] >= 0 THEN
							Internal.Pair.Name								:= DINT_TO_STRING(Internal.DepthArrayIdx[Internal.Depth]);
							Internal.DepthArrayIdx[Internal.Depth] 			:= Internal.DepthArrayIdx[Internal.Depth] + 1;
							Internal.InValue								:= TRUE;
						END_IF;
					ELSIF TC_Find_S(pBuffer+Internal.i,ADR(':')) >= 0 THEN
						// Value is next
						Internal.InValue									:= TRUE;
						Internal.Marker										:= Internal.i+1;
					ELSIF TC_Find_S(pBuffer+Internal.i,ADR(']')) >= 0 THEN
						IF Internal.InValue THEN
							Internal.InValue								:= FALSE;
							IF Internal.i <> 0 AND UDINT_TO_DINT(Internal.Marker) < Internal.i THEN
								IF (Internal.i - UDINT_TO_DINT(Internal.Marker)) < SIZEOF(Internal.Pair.Value) THEN
									brsmemcpy(ADR(Internal.Pair.Value),pBuffer+Internal.Marker,(Internal.i-Internal.Marker));
								ELSE
									brsmemcpy(ADR(Internal.Pair.Value),pBuffer+Internal.Marker,SIZEOF(Internal.Pair.Value)-1);
								END_IF;
								Internal.i 									:= Internal.i-1; 							// Go back one step to hit the bracket close again.
								Internal.Send								:= TRUE;
							ELSE
								Error										:= TRUE;
								EXIT;
							END_IF;
						ELSE
							Internal.DepthArrayIdx[Internal.Depth]			:= -1;
							Internal.Pair.Name								:= Internal.DepthIDs[Internal.Depth];
							Internal.DepthIDs[Internal.Depth]				:= '';
							Internal.Pair.Value								:= ']';
							Internal.Send									:= TRUE;
							IF Internal.Depth = 0 THEN
								Error										:= TRUE;
								EXIT;
							ELSE
								Internal.Depth								:= Internal.Depth - 1;
							END_IF;
						END_IF;
					ELSIF TC_Find_S(pBuffer+Internal.i,ADR('}')) >= 0 THEN
						IF Internal.InValue THEN
							Internal.InValue								:= FALSE;
							IF Internal.i <> 0 AND UDINT_TO_DINT(Internal.Marker) < Internal.i THEN
								IF (Internal.i - UDINT_TO_DINT(Internal.Marker)) < SIZEOF(Internal.Pair.Value) THEN
									brsmemcpy(ADR(Internal.Pair.Value),pBuffer+Internal.Marker,(Internal.i-Internal.Marker));
								ELSE
									brsmemcpy(ADR(Internal.Pair.Value),pBuffer+Internal.Marker,SIZEOF(Internal.Pair.Value)-1);
								END_IF;
								Internal.i 									:= Internal.i-1; 							// Go back one step to hit the bracket close again.
								Internal.Send								:= TRUE;
							ELSE
								Error										:= TRUE;
								EXIT;
							END_IF;
						ELSE
							Internal.DepthArrayIdx[Internal.Depth]			:= -1;
							Internal.Pair.Name								:= Internal.DepthIDs[Internal.Depth];
							Internal.DepthIDs[Internal.Depth]				:= '';
							Internal.Pair.Value								:= '}';
							Internal.Send									:= TRUE;
							IF Internal.Depth = 0 THEN
								Error										:= TRUE;
								EXIT;
							ELSE
								Internal.Depth								:= Internal.Depth - 1;
							END_IF;
						END_IF;
					ELSIF TC_Find_S(pBuffer+Internal.i,ADR(',')) >= 0 THEN
						IF Internal.InValue THEN
							Internal.InValue								:= FALSE;
							Internal.Send 									:= TRUE;
							IF Internal.i <> 0 AND UDINT_TO_DINT(Internal.Marker) < Internal.i THEN
								IF (Internal.i - UDINT_TO_DINT(Internal.Marker)) < SIZEOF(Internal.Pair.Value) THEN
									brsmemcpy(ADR(Internal.Pair.Value),pBuffer+Internal.Marker,(Internal.i-Internal.Marker));
								ELSE
									brsmemcpy(ADR(Internal.Pair.Value),pBuffer+Internal.Marker,SIZEOF(Internal.Pair.Value)-1);
								END_IF;
							ELSE
								Error										:= TRUE;
								EXIT;
							END_IF;
						END_IF;
					ELSIF TC_Find_S(pBuffer+Internal.i,ADR(' ')) >= 0 OR TC_Find_S(pBuffer+Internal.i,ADR('	')) >= 0 OR TC_Find_S(pBuffer+Internal.i,ADR('$r')) >= 0 OR TC_Find_S(pBuffer+Internal.i,ADR('$n')) >= 0 THEN //Whitespace
						IF NOT Internal.InValueNonWhiteFound THEN
							Internal.Marker									:= Internal.i+1;
						ELSIF Internal.InValue THEN
							Internal.InValue								:= FALSE;
							Internal.InValueNonWhiteFound					:= FALSE;
							IF Internal.i <> 0 AND UDINT_TO_DINT(Internal.Marker) < Internal.i THEN
								IF (Internal.i - UDINT_TO_DINT(Internal.Marker)) < SIZEOF(Internal.Pair.Value) THEN
									brsmemcpy(ADR(Internal.Pair.Value),pBuffer+Internal.Marker,(Internal.i-Internal.Marker));
								ELSE
									brsmemcpy(ADR(Internal.Pair.Value),pBuffer+Internal.Marker,SIZEOF(Internal.Pair.Value)-1);
								END_IF;
							ELSE
								Error										:= TRUE;
								EXIT;
							END_IF;
							Internal.Send 									:= TRUE;
						END_IF;
					ELSIF Internal.InValue OR Internal.DepthArrayIdx[Internal.Depth] >= 0 THEN
						Internal.InValue									:= TRUE;
						Internal.InValueNonWhiteFound						:= TRUE;
					END_IF;
				ELSIF Internal.QuoteIsDouble THEN 																		//Inside Double Quotes
					IF TC_Find_S(pBuffer+Internal.i,ADR('"')) >= 0 THEN
						IF Internal.InValue THEN
							Internal.InValue								:= FALSE;
							Internal.Send 									:= TRUE;
							IF Internal.i <> 0 AND UDINT_TO_DINT(Internal.Marker) < Internal.i THEN
								IF (Internal.i - UDINT_TO_DINT(Internal.Marker)) < SIZEOF(Internal.Pair.Value) THEN
									IF NoQuotes THEN
										brsmemcpy(ADR(Internal.Pair.Value),pBuffer+Internal.Marker,(Internal.i-Internal.Marker));
									ELSE
										brsmemcpy(ADR(Internal.Pair.Value),ADR('"'),1);
										brsmemcpy(ADR(Internal.Pair.Value)+1,pBuffer+Internal.Marker,(Internal.i-Internal.Marker));
										brsmemcpy(ADR(Internal.Pair.Value)+1+(Internal.i-Internal.Marker),ADR('"'),1);
									END_IF;
								ELSE
									IF NoQuotes THEN
										brsmemcpy(ADR(Internal.Pair.Value),pBuffer+Internal.Marker,SIZEOF(Internal.Pair.Value)-1);
									ELSE
										brsmemcpy(ADR(Internal.Pair.Value),ADR('"'),1);
										brsmemcpy(ADR(Internal.Pair.Value)+1,pBuffer+Internal.Marker,SIZEOF(Internal.Pair.Value)-3);
										brsmemcpy(ADR(Internal.Pair.Value)+SIZEOF(Internal.Pair.Value)-1,ADR('"'),1);
									END_IF;
								END_IF;
							ELSIF Internal.i <> 0 AND UDINT_TO_DINT(Internal.Marker) = Internal.i THEN
								IF NoQuotes THEN
									//Nothing
								ELSE
									brsmemcpy(ADR(Internal.Pair.Value),ADR('""'),2);
								END_IF;
							ELSE
								Error										:= TRUE;
								EXIT;
							END_IF;
						ELSE
							IF Internal.i <> 0 AND UDINT_TO_DINT(Internal.Marker) < Internal.i THEN
								IF (Internal.i - UDINT_TO_DINT(Internal.Marker)) < SIZEOF(Internal.Pair.Name) THEN
									brsmemcpy(ADR(Internal.Pair.Name),pBuffer+Internal.Marker,(Internal.i-Internal.Marker));
								ELSE
									brsmemcpy(ADR(Internal.Pair.Name),pBuffer+Internal.Marker,SIZEOF(Internal.Pair.Name)-1);
								END_IF;
							ELSE
								Error										:= TRUE;
								EXIT;
							END_IF;
						END_IF;
						Internal.InQuote 									:= FALSE;
						Internal.QuoteIsDouble 								:= FALSE;
					END_IF;
				ELSE 																									//Inside Single Quotes
					IF TC_Find_S(pBuffer+Internal.i,ADR('$'')) >= 0 THEN
						IF Internal.InValue THEN
							Internal.InValue								:= FALSE;
							Internal.Send 									:= TRUE;
							IF Internal.i <> 0 AND UDINT_TO_DINT(Internal.Marker) < Internal.i THEN
								IF (Internal.i - UDINT_TO_DINT(Internal.Marker)) < SIZEOF(Internal.Pair.Value) THEN
									IF NoQuotes THEN
										brsmemcpy(ADR(Internal.Pair.Value),pBuffer+Internal.Marker,(Internal.i-Internal.Marker));
									ELSE
										brsmemcpy(ADR(Internal.Pair.Value),ADR('$''),1);
										brsmemcpy(ADR(Internal.Pair.Value)+1,pBuffer+Internal.Marker,(Internal.i-Internal.Marker));
										brsmemcpy(ADR(Internal.Pair.Value)+1+(Internal.i-Internal.Marker),ADR('$''),1);
									END_IF;
								ELSE
									IF NoQuotes THEN
										brsmemcpy(ADR(Internal.Pair.Value),pBuffer+Internal.Marker,SIZEOF(Internal.Pair.Value)-1);
									ELSE
										brsmemcpy(ADR(Internal.Pair.Value),ADR('$''),1);
										brsmemcpy(ADR(Internal.Pair.Value)+1,pBuffer+Internal.Marker,SIZEOF(Internal.Pair.Value)-3);
										brsmemcpy(ADR(Internal.Pair.Value)+SIZEOF(Internal.Pair.Value)-1,ADR('$''),1);
									END_IF;
								END_IF;
							ELSIF Internal.i <> 0 AND UDINT_TO_DINT(Internal.Marker) = Internal.i THEN
								IF NoQuotes THEN
									//Nothing
								ELSE
									brsmemcpy(ADR(Internal.Pair.Value),ADR('$'$''),2);
								END_IF;
							ELSE
								Error										:= TRUE;
								EXIT;
							END_IF;
						ELSE
							IF Internal.i <> 0 AND UDINT_TO_DINT(Internal.Marker) < Internal.i THEN
								IF (Internal.i - UDINT_TO_DINT(Internal.Marker)) < SIZEOF(Internal.Pair.Name) THEN
									brsmemcpy(ADR(Internal.Pair.Name),pBuffer+Internal.Marker,(Internal.i-Internal.Marker));
								ELSE
									brsmemcpy(ADR(Internal.Pair.Name),pBuffer+Internal.Marker,SIZEOF(Internal.Pair.Name)-1);
								END_IF;
							ELSE
								Error										:= TRUE;
								EXIT;
							END_IF;
						END_IF;
						Internal.InQuote 									:= FALSE;
						Internal.QuoteIsDouble 								:= FALSE;
					END_IF;
				END_IF;
				IF Internal.Send THEN
					Internal.Send											:= FALSE;
					IF Internal.Idx >= 0 AND Internal.Idx <= MAX_JSON_PARSE_PAIR_IDX THEN
						brsmemcpy(pPairs+Internal.Idx*SIZEOF(Internal.Pair),ADR(Internal.Pair),SIZEOF(Internal.Pair));
						brsmemset(ADR(Internal.Pair),0,SIZEOF(Internal.Pair));
						Internal.InQuote									:= FALSE;
						Internal.InValue									:= FALSE;
						Internal.InValueNonWhiteFound						:= FALSE;
						Internal.Marker										:= 0;
						Internal.Idx										:= Internal.Idx + 1;
					ELSE
						Error												:= TRUE;
						EXIT;
					END_IF;
				END_IF;
			END_FOR;
			IF NOT Error THEN
				Done														:= TRUE;
			END_IF;
		END_IF;
	ELSE
		Done																:= FALSE;
		Error																:= FALSE;
		brsmemset(ADR(Internal),0,SIZEOF(Internal));
	END_IF;

END_FUNCTION_BLOCK
```

#### TC_JSON_PairsToJSON.st
```iecst
(* Takes Value Pairs and packs into a JSON String *)
FUNCTION_BLOCK TC_JSON_PairsToJSON
	IF Enable THEN
		IF NOT Internal.Enabled THEN
			brsmemset(ADR(Internal),0,SIZEOF(Internal));
			brsmemset(pBuffer,0,BufferSIZEOF);
			TC_brsstrcat(pBuffer,ADR('$r$n'),BufferSIZEOF);
			Internal.DepthArrayIdx[0]										:= -1;
			Internal.Enabled												:= TRUE;
		END_IF;
		IF Error OR Done THEN
			// Do Nothing, Enable must be toggled to parse again
		ELSE
			FOR Internal.i := 0 TO MAX_JSON_PARSE_PAIR_IDX DO
				brsmemcpy(ADR(Internal.Pair),pPairs+SIZEOF(Internal.Pair)*Internal.i,SIZEOF(Internal.Pair));
				IF Internal.Pair.Name = '' AND Internal.Pair.Value = '' THEN
					TC_brsstrcat(pBuffer,ADR('$r$n'),BufferSIZEOF);
					Done													:= TRUE;
					EXIT;
				ELSIF Internal.i = MAX_JSON_PARSE_PAIR_IDX AND Internal.Pair.Value <> '}' THEN
					Error													:= TRUE;
					EXIT;
				ELSE
					IF Internal.Pair.Value = '{' THEN
						IF Internal.Depth <= MAX_JSON_PARSE_DEPTH_IDX THEN
							Internal.Depth 									:= Internal.Depth + 1;
							Internal.DepthArrayIdx[Internal.Depth]			:= -1;
							IF Internal.DepthArrayIdx[Internal.Depth-1] >= 0 OR Internal.i = 0 THEN
								TC_brsstrcat(pBuffer,ADR('{'),BufferSIZEOF);
							ELSE
								TC_brsstrcat(pBuffer,ADR('"'),BufferSIZEOF);
								TC_brsstrcat(pBuffer,ADR(Internal.Pair.Name),BufferSIZEOF);
								TC_brsstrcat(pBuffer,ADR('": {'),BufferSIZEOF);
							END_IF;
							IF Internal.i <> MAX_JSON_PARSE_PAIR_IDX THEN
								brsmemcpy(ADR(Internal.Pair),pPairs+SIZEOF(Internal.Pair)*(Internal.i+1),SIZEOF(Internal.Pair));
								IF Internal.Pair.Value <> '}' THEN // Check next element to detect empty object condition
									TC_brsstrcat(pBuffer,ADR('$r$n'),BufferSIZEOF);
									FOR Internal.j := 0 TO (Internal.Depth-1)*2+1 DO
										TC_brsstrcat(pBuffer,ADR(' '),BufferSIZEOF);
									END_FOR;
								END_IF;
								brsmemcpy(ADR(Internal.Pair),pPairs+SIZEOF(Internal.Pair)*Internal.i,SIZEOF(Internal.Pair));
							END_IF;
						ELSE
							Error											:= TRUE;
							EXIT;
						END_IF;
					ELSIF Internal.Pair.Value = '}' THEN
						Internal.DepthArrayIdx[Internal.Depth]			:= -1;
						IF Internal.Depth = 0 THEN
							Error										:= TRUE;
							EXIT;
						ELSE
							Internal.Depth								:= Internal.Depth - 1;
						END_IF;
						TC_brsstrcat(pBuffer,ADR('}'),BufferSIZEOF);
						IF Internal.i <> MAX_JSON_PARSE_PAIR_IDX THEN
							brsmemcpy(ADR(Internal.Pair),pPairs+SIZEOF(Internal.Pair)*(Internal.i+1),SIZEOF(Internal.Pair));
							IF Internal.Pair.Value = '' AND Internal.Pair.Value = '' THEN

							ELSIF Internal.Pair.Value <> ']' AND Internal.Pair.Value <> '}' THEN
								TC_brsstrcat(pBuffer,ADR(','),BufferSIZEOF);
								TC_brsstrcat(pBuffer,ADR('$r$n'),BufferSIZEOF);
								FOR Internal.j := 0 TO (Internal.Depth-1)*2+1 DO
									TC_brsstrcat(pBuffer,ADR(' '),BufferSIZEOF);
								END_FOR;
							ELSE
								TC_brsstrcat(pBuffer,ADR('$r$n'),BufferSIZEOF);
								IF Internal.Depth >= 2 THEN
									FOR Internal.j := 0 TO (Internal.Depth-2)*2+1 DO
										TC_brsstrcat(pBuffer,ADR(' '),BufferSIZEOF);
									END_FOR;
								END_IF;
							END_IF;
							brsmemcpy(ADR(Internal.Pair),pPairs+SIZEOF(Internal.Pair)*Internal.i,SIZEOF(Internal.Pair));
						END_IF;
					ELSIF Internal.Pair.Value = '[' THEN
						IF Internal.Depth <= MAX_JSON_PARSE_DEPTH_IDX THEN
							Internal.Depth 									:= Internal.Depth + 1;
							Internal.DepthArrayIdx[Internal.Depth]			:= 0;
							IF Internal.DepthArrayIdx[Internal.Depth-1] >= 0 OR Internal.i = 0 THEN
								TC_brsstrcat(pBuffer,ADR('['),BufferSIZEOF);
							ELSE
								TC_brsstrcat(pBuffer,ADR('"'),BufferSIZEOF);
								TC_brsstrcat(pBuffer,ADR(Internal.Pair.Name),BufferSIZEOF);
								TC_brsstrcat(pBuffer,ADR('": ['),BufferSIZEOF);
							END_IF;
							IF Internal.i <> MAX_JSON_PARSE_PAIR_IDX THEN
								brsmemcpy(ADR(Internal.Pair),pPairs+SIZEOF(Internal.Pair)*(Internal.i+1),SIZEOF(Internal.Pair));
								IF Internal.Pair.Value = '[' OR Internal.Pair.Value = '{' THEN
									TC_brsstrcat(pBuffer,ADR('$r$n'),BufferSIZEOF);
									IF Internal.Depth >= 1 THEN
										FOR Internal.j := 0 TO (Internal.Depth-1)*2+1 DO
											TC_brsstrcat(pBuffer,ADR(' '),BufferSIZEOF);
										END_FOR;
									END_IF;
								END_IF;
								brsmemcpy(ADR(Internal.Pair),pPairs+SIZEOF(Internal.Pair)*Internal.i,SIZEOF(Internal.Pair));
							END_IF;
						ELSE
							Error											:= TRUE;
							EXIT;
						END_IF;
					ELSIF Internal.Pair.Value = ']' THEN
						Internal.DepthArrayIdx[Internal.Depth]			:= -1;
						IF Internal.Depth = 0 THEN
							Error										:= TRUE;
							EXIT;
						ELSE
							Internal.Depth								:= Internal.Depth - 1;
						END_IF;
						TC_brsstrcat(pBuffer,ADR(']'),BufferSIZEOF);
						IF Internal.i <> MAX_JSON_PARSE_PAIR_IDX THEN
							brsmemcpy(ADR(Internal.Pair),pPairs+SIZEOF(Internal.Pair)*(Internal.i+1),SIZEOF(Internal.Pair));
							IF Internal.Pair.Value = '' AND Internal.Pair.Value = '' THEN

							ELSIF Internal.Pair.Value <> ']' AND Internal.Pair.Value <> '}' THEN
								TC_brsstrcat(pBuffer,ADR(','),BufferSIZEOF);
								TC_brsstrcat(pBuffer,ADR('$r$n'),BufferSIZEOF);
								FOR Internal.j := 0 TO (Internal.Depth-1)*2+1 DO
									TC_brsstrcat(pBuffer,ADR(' '),BufferSIZEOF);
								END_FOR;
							ELSE
								TC_brsstrcat(pBuffer,ADR('$r$n'),BufferSIZEOF);
								IF Internal.Depth >= 2 THEN
									FOR Internal.j := 0 TO (Internal.Depth-2)*2+1 DO
										TC_brsstrcat(pBuffer,ADR(' '),BufferSIZEOF);
									END_FOR;
								END_IF;
							END_IF;
							brsmemcpy(ADR(Internal.Pair),pPairs+SIZEOF(Internal.Pair)*Internal.i,SIZEOF(Internal.Pair));
						END_IF;
					ELSE
						IF Internal.DepthArrayIdx[Internal.Depth] >= 0 THEN
							TC_brsstrcat(pBuffer,ADR(Internal.Pair.Value),BufferSIZEOF);
							IF Internal.i <> MAX_JSON_PARSE_PAIR_IDX THEN
								brsmemcpy(ADR(Internal.Pair),pPairs+SIZEOF(Internal.Pair)*(Internal.i+1),SIZEOF(Internal.Pair));
								IF Internal.Pair.Value <> ']' AND Internal.Pair.Value <> '}' THEN
									TC_brsstrcat(pBuffer,ADR(', '),BufferSIZEOF);
								END_IF;
								brsmemcpy(ADR(Internal.Pair),pPairs+SIZEOF(Internal.Pair)*Internal.i,SIZEOF(Internal.Pair));
							END_IF;
						ELSE
							TC_brsstrcat(pBuffer,ADR('"'),BufferSIZEOF);
							TC_brsstrcat(pBuffer,ADR(Internal.Pair.Name),BufferSIZEOF);
							TC_brsstrcat(pBuffer,ADR('": '),BufferSIZEOF);
							TC_brsstrcat(pBuffer,ADR(Internal.Pair.Value),BufferSIZEOF);
							IF Internal.i <> MAX_JSON_PARSE_PAIR_IDX THEN
								brsmemcpy(ADR(Internal.Pair),pPairs+SIZEOF(Internal.Pair)*(Internal.i+1),SIZEOF(Internal.Pair));
								IF Internal.Pair.Value <> ']' AND Internal.Pair.Value <> '}' THEN
									TC_brsstrcat(pBuffer,ADR(','),BufferSIZEOF);
									TC_brsstrcat(pBuffer,ADR('$r$n'),BufferSIZEOF);
									FOR Internal.j := 0 TO (Internal.Depth-1)*2+1 DO
										TC_brsstrcat(pBuffer,ADR(' '),BufferSIZEOF);
									END_FOR;
								ELSE
									TC_brsstrcat(pBuffer,ADR('$r$n'),BufferSIZEOF);
									IF Internal.Depth >= 2 THEN
										FOR Internal.j := 0 TO (Internal.Depth-2)*2+1 DO
											TC_brsstrcat(pBuffer,ADR(' '),BufferSIZEOF);
										END_FOR;
									END_IF;
								END_IF;
								brsmemcpy(ADR(Internal.Pair),pPairs+SIZEOF(Internal.Pair)*Internal.i,SIZEOF(Internal.Pair));
							END_IF;
						END_IF;
					END_IF;
				END_IF;
			END_FOR;
		END_IF;
	ELSE
		Done																:= FALSE;
		Error																:= FALSE;
		brsmemset(ADR(Internal),0,SIZEOF(Internal));
	END_IF;

END_FUNCTION_BLOCK
```

### Library Logical/Libraries/TC_Seq (IEC)
Depends on: TC_General, AsBrStr, brsystem, TC_JSON

#### Types.typ - Exported data types
```iecst
TYPE
	TC_Seq_Par_Element_typ : 	STRUCT
		Name : STRING[255];
		GenVar : TC_Seq_GenVar_typ;
	END_STRUCT;
	TC_Seq_GenVar_typ : 	STRUCT
		Select : TC_SEQ_PAR_SELECT_ENUM;
		VarBOOL : BOOL;
		VarSINT : SINT;
		VarUSINT : USINT;
		VarINT : INT;
		VarUINT : UINT;
		VarDINT : DINT;
		VarUDINT : UDINT;
		VarREAL : REAL;
		VarLREAL : LREAL;
		VarTIME : TIME;
		VarDT : DATE_AND_TIME;
		VarSTRING : STRING[MAX_JSON_PARSE_VALUE_LEN];
		VarSTRING_ADR : UDINT;
		VarADR : UDINT;
		VarENUM : DINT;
		VarENUM_STRING : STRING[32];
	END_STRUCT;
	TC_Seq_ESS_Internal_typ : 	STRUCT
		PvRoot : STRING[255];
		PvName : STRING[255];
		PvValue : STRING[32];
		IdxString : STRING[32];
		PvLen : UDINT;
		PvAddress : UDINT;
		DataLen : UDINT;
		Datatype : UDINT;
		Dimension : UINT;
		Status : UINT;
		i : DINT;
	END_STRUCT;
	TC_Seq_Handler_Buffer_typ : 	STRUCT
		Type : TC_SEQ_TYPE_ENUM;
		Json : STRING[MAX_TC_SEQ_JSON_STRING_LEN];
		Time : LREAL;
		WaitPvAddress : UDINT;
		UID : DINT;
		Status : DINT;
	END_STRUCT;
	TC_Seq_JsonToElem_Internal_typ : 	STRUCT
		idx : DINT;
		i : DINT;
		TC_JSON_Parse_0 : TC_JSON_Parse;
		JSONPairs : ARRAY[0..MAX_JSON_PARSE_PAIR_IDX]OF TC_JSON_Parse_Pair_typ;
		Element : TC_Seq_Handler_Buffer_typ;
		EnumNameString_Ident : STRING[32];
		EnumValueString_Ident : STRING[32];
		IdentIdxString : STRING[32];
		IdentIdx : DINT;
		EnumNameString_Inst : STRING[32];
		EnumValueString_Inst : STRING[32];
		InstIdxString : STRING[32];
		InstIdx : DINT;
		DriverRoot : STRING[255];
		PvName : STRING[255];
		PvNameSub : STRING[255];
		PvLen : UDINT;
		DataLen : UDINT;
		ParValue : STRING[MAX_JSON_PARSE_VALUE_LEN];
		ParDataType : STRING[2];
		Datatype : UDINT;
		Dimension : UINT;
		ParPvAddress : ARRAY[0..MAX_TC_SEQ_PAR_IDX]OF UDINT;
		WaitPvAddress : UDINT;
		CmdPvAddress : UDINT;
		PvAddress : UDINT;
		Status : UINT;
		ParElement : ARRAY[0..MAX_JSON_PARSE_PAIR_IDX]OF TC_Seq_Par_Element_typ;
		Driver : STRING[32];
		Ident : STRING[32];
		Inst : STRING[32];
		Sev : DINT;
		Enable : BOOL;
		ParDone : BOOL;
		Par : STRING[MAX_TC_SEQ_PAR_STRING_LEN];
	END_STRUCT;
	TC_Seq_Generic_Internal_typ : 	STRUCT
		i : DINT;
	END_STRUCT;
	TC_Seq_Handler_Internal_typ : 	STRUCT
		i : DINT;
		ErrorID : DINT;
		CTON_0 : CTON;
		LastState : TC_SEQ_HANDLER_STATE_ENUM;
		State : TC_SEQ_HANDLER_STATE_ENUM;
		CurrentWait : DINT;
		TempJson : STRING[MAX_TC_SEQ_JSON_STRING_LEN];
		CurrentBuffer : TC_Seq_Handler_Buffer_typ;
		RTInfo_0 : RTInfo;
		TimeIncrement : LREAL;
		CurrentDelay : LREAL;
		Status : DINT;
	END_STRUCT;
	TC_Seq_Handler_Out_typ : 	STRUCT
		Status : TC_Seq_Handler_Out_Status_typ;
		Buffer : TC_Seq_Handler_Out_Buffer_typ;
	END_STRUCT;
	TC_Seq_Handler_Out_Buffer_typ : 	STRUCT
		Last : ARRAY[0..MAX_TC_SEQ_BUFFER_LAST_IDX]OF TC_Seq_Handler_Buffer_typ;
		Current : TC_Seq_Handler_Buffer_typ;
	END_STRUCT;
	TC_Seq_Handler_Out_Status_typ : 	STRUCT
		Remaining : LREAL;
		Elapsed : LREAL;
		InReset : BOOL;
		Paused : BOOL;
		Ready : BOOL;
		Processing : BOOL;
		Error : BOOL;
		ErrorID : DINT;
		CurrentState : STRING[32];
		Timeout : BOOL;
		Interrupt : BOOL;
	END_STRUCT;
	TC_Seq_Buffer_Info_typ : 	STRUCT
		pUID : UDINT;
		pBuffer : UDINT;
	END_STRUCT;
	TC_SEQ_HANDLER_STATE_ENUM :
		( (*ENUM_STRING*)
		TC_SEQ_HANDLER_RESET,
		TC_SEQ_HANDLER_EVAL,
		TC_SEQ_HANDLER_CMD,
		TC_SEQ_HANDLER_WAIT,
		TC_SEQ_HANDLER_DELAY,
		TC_SEQ_HANDLER_INTERRUPT,
		TC_SEQ_HANDLER_ERROR
		);
	TC_SEQ_WAIT_ENUM :
		( (*ENUM_STRING*)
		TC_SEQ_WAIT_FALSE,
		TC_SEQ_WAIT_TRUE,
		TC_SEQ_WAIT_INTERRUPT,
		TC_SEQ_WAIT_ERROR
		);
	TC_SEQ_TYPE_ENUM :
		( (*ENUM_STRING*)
		TC_SEQ_TYPE_NONE,
		TC_SEQ_TYPE_CMD,
		TC_SEQ_TYPE_WAIT,
		TC_SEQ_TYPE_MON,
		TC_SEQ_TYPE_DELAY,
		TC_SEQ_TYPE_BREAK
		);
	TC_SEQ_PAR_SELECT_ENUM :
		( (*ENUM_STRING*)
		TC_SEQ_PAR_SELECT_NULL,
		TC_SEQ_PAR_SELECT_BOOL,
		TC_SEQ_PAR_SELECT_INT,
		TC_SEQ_PAR_SELECT_USINT,
		TC_SEQ_PAR_SELECT_SINT,
		TC_SEQ_PAR_SELECT_UINT,
		TC_SEQ_PAR_SELECT_DINT,
		TC_SEQ_PAR_SELECT_UDINT,
		TC_SEQ_PAR_SELECT_REAL,
		TC_SEQ_PAR_SELECT_LREAL,
		TC_SEQ_PAR_SELECT_TIME,
		TC_SEQ_PAR_SELECT_DT,
		TC_SEQ_PAR_SELECT_ENUMNAME,
		TC_SEQ_PAR_SELECT_STRING,
		TC_SEQ_PAR_SELECT_STRINGADR,
		TC_SEQ_PAR_SELECT_STRINGLEN,
		TC_SEQ_PAR_SELECT_WSTRINGADR,
		TC_SEQ_PAR_SELECT_WSTRINGLEN,
		TC_SEQ_PAR_SELECT_ADR,
		TC_SEQ_PAR_SELECT_PTR
		);
END_TYPE
```

#### Constants.var - Exported constants
```iecst
VAR CONSTANT
	MAX_TC_SEQ_CMD_IDX : DINT := 99;
	MAX_TC_SEQ_WAIT_IDX : DINT := 99;
	MAX_TC_SEQ_BUFFER_IDX : DINT := 399;
	MAX_TC_SEQ_BUFFER_LAST_IDX : DINT := 4;
	MAX_TC_SEQ_PAR_IDX : DINT := 19;
	MAX_TC_SEQ_JSON_STRING_LEN : DINT := 1000;
	MAX_TC_SEQ_PAR_STRING_LEN : DINT := 500;
	MAX_TC_SEQ_META_STRING_LEN : DINT := 32;
	MAX_TC_SEQ_SYNC_IDX : DINT := 10;
END_VAR
```

#### TC_Seq.fun - Exported functions and function blocks
```iecst
{REDUND_ERROR} FUNCTION_BLOCK TC_Seq_Handler (*Sequence Handler*) (*$GROUP=User,$CAT=User,$GROUPICON=User.png,$CATICON=User.png*)
	VAR_INPUT
		Enable : BOOL;
		Reset : BOOL;
		ErrorReset : BOOL;
		ClearBuffer : BOOL;
		ForceNext : BOOL;
		Pause : BOOL;
		pJsonArray : UDINT;
	END_VAR
	VAR_OUTPUT
		Out : TC_Seq_Handler_Out_typ;
	END_VAR
	VAR
		Internal : TC_Seq_Handler_Internal_typ;
	END_VAR
END_FUNCTION_BLOCK

{REDUND_ERROR} FUNCTION TC_Seq_EnumStringSearch : DINT (*Returns a negative value if not found*) (*$GROUP=User,$CAT=User,$GROUPICON=User.png,$CATICON=User.png*)
	VAR_INPUT
		EnumNameSTRING : STRING[32]; (*STRING*)
		EnumValueSTRING : STRING[32]; (*STRING*)
	END_VAR
	VAR
		Internal : TC_Seq_ESS_Internal_typ;
	END_VAR
END_FUNCTION

{REDUND_ERROR} FUNCTION TC_Seq_JsonToElem : DINT (* *) (*$GROUP=User,$CAT=User,$GROUPICON=User.png,$CATICON=User.png*)
	VAR_INPUT
		pJsonString : UDINT;
		pElement : UDINT;
	END_VAR
	VAR
		Internal : TC_Seq_JsonToElem_Internal_typ;
	END_VAR
END_FUNCTION

{REDUND_ERROR} FUNCTION TC_Seq_Add : DINT (* *) (*$GROUP=User,$CAT=User,$GROUPICON=User.png,$CATICON=User.png*)
	VAR_INPUT
		pJsonArray : UDINT;
		pJson : UDINT;
	END_VAR
	VAR
		Internal : TC_Seq_Generic_Internal_typ;
	END_VAR
END_FUNCTION

{REDUND_ERROR} FUNCTION TC_Seq_AddFront : DINT (* *) (*$GROUP=User,$CAT=User,$GROUPICON=User.png,$CATICON=User.png*)
	VAR_INPUT
		pJsonArray : UDINT;
		pJson : UDINT;
	END_VAR
	VAR
		Internal : TC_Seq_Generic_Internal_typ;
	END_VAR
END_FUNCTION
```

#### TC_Seq_Handler.st
```iecst
(* Sequence Handler *)
FUNCTION_BLOCK TC_Seq_Handler
	IF NOT Enable OR Reset OR pJsonArray = 0 THEN
		Internal.State									:= TC_SEQ_HANDLER_RESET;
	ELSIF ClearBuffer THEN
		brsmemset(pJsonArray,0,SIZEOF(Internal.TempJson)*DINT_TO_UDINT((MAX_TC_SEQ_BUFFER_IDX+1)));
	END_IF;
	brsmemset(ADR(Out.Status),0,SIZEOF(Out.Status));
	CASE Internal.State OF
		TC_SEQ_HANDLER_RESET:
			brsmemset(ADR(Internal),0,SIZEOF(Internal));
			brsmemset(ADR(Out),0,SIZEOF(Out));
			Out.Status.CurrentState						:= 'TC_SEQ_HANDLER_RESET';
			IF Enable AND NOT Reset THEN
				Internal.State							:= TC_SEQ_HANDLER_EVAL;
			END_IF;
		TC_SEQ_HANDLER_EVAL:
			Out.Status.CurrentState						:= 'TC_SEQ_HANDLER_EVAL';
			Out.Status.Processing						:= TRUE;
			brsmemset(ADR(Internal.CurrentBuffer),0,SIZEOF(Internal.CurrentBuffer));
			brsmemset(ADR(Internal.TempJson),0,SIZEOF(Internal.TempJson));
			IF Pause THEN
				Out.Status.Processing					:= FALSE;
				Out.Status.Paused						:= TRUE;
			ELSE
				FOR Internal.i := MAX_TC_SEQ_BUFFER_IDX TO 0 BY -1 DO
					brsmemcpy(ADR(Internal.TempJson),pJsonArray+Internal.i*SIZEOF(Internal.TempJson),SIZEOF(Internal.TempJson));
					IF Internal.TempJson <> '' THEN
						Internal.Status := TC_Seq_JsonToElem(ADR(Internal.TempJson),ADR(Internal.CurrentBuffer));
						IF Internal.Status = 0 THEN
							brsmemset(pJsonArray+Internal.i*SIZEOF(Internal.TempJson),0,SIZEOF(Internal.TempJson));
						ELSE
							Out.Status.ErrorID 	:= Internal.Status;
							Out.Status.Error 	:= TRUE;
						END_IF;
						EXIT;
					END_IF;
				END_FOR;
				IF NOT Out.Status.Error THEN
					CASE Internal.CurrentBuffer.Type OF
						TC_SEQ_TYPE_NONE:
							Out.Status.Processing			:= FALSE;
							Out.Status.Ready				:= TRUE;
						TC_SEQ_TYPE_CMD:
							Out.Status.Processing			:= TRUE;
							IF Internal.CurrentBuffer.Time <> 0 THEN
								Internal.State				:= TC_SEQ_HANDLER_CMD;
							END_IF;
						TC_SEQ_TYPE_WAIT:
							Out.Status.Processing			:= TRUE;
							Internal.State					:= TC_SEQ_HANDLER_WAIT;
						TC_SEQ_TYPE_MON:
							Out.Status.Processing			:= TRUE;
						TC_SEQ_TYPE_DELAY:
							Out.Status.Processing			:= TRUE;
							IF Internal.CurrentBuffer.Time > 0.0 THEN
								Internal.RTInfo_0(enable := TRUE);
								Internal.TimeIncrement		:= UDINT_TO_LREAL(Internal.RTInfo_0.cycle_time)/1000000.0;
								Internal.CurrentDelay		:= Internal.CurrentBuffer.Time - Internal.TimeIncrement*3.0;
								IF Internal.CurrentDelay >= 0.0 THEN
									Internal.State			:= TC_SEQ_HANDLER_DELAY;
								END_IF;
							END_IF;
						TC_SEQ_TYPE_BREAK:
							Out.Status.Processing			:= TRUE;
							Internal.State					:= TC_SEQ_HANDLER_EVAL;
						ELSE
							Out.Status.Processing			:= FALSE;
							Out.Status.Error				:= TRUE;
							Internal.ErrorID.28				:= 1;
							Internal.State					:= TC_SEQ_HANDLER_ERROR;
					END_CASE;
				END_IF;
			END_IF;
		TC_SEQ_HANDLER_CMD:
			Out.Status.CurrentState						:= 'TC_SEQ_HANDLER_CMD';
			Out.Status.Processing						:= TRUE;
			Internal.CTON_0.IN							:= TRUE;
			Internal.CTON_0.PT							:= LREAL_TO_TIME(Internal.CurrentBuffer.Time*1000.0);
			Internal.CTON_0.PAUSE						:= FALSE;
			Internal.State								:= TC_SEQ_HANDLER_EVAL;
		TC_SEQ_HANDLER_WAIT:
			Out.Status.CurrentState						:= 'TC_SEQ_HANDLER_WAIT';
			Out.Status.Processing						:= TRUE;
			Internal.CTON_0.IN							:= TRUE;
			Internal.CTON_0.PT							:= LREAL_TO_TIME(Internal.CurrentBuffer.Time*1000.0);
			Internal.CTON_0.PAUSE						:= FALSE;
			brsmemcpy(ADR(Internal.CurrentWait),Internal.CurrentBuffer.WaitPvAddress,SIZEOF(Internal.CurrentWait));
			IF ForceNext = TRUE THEN
				Internal.State							:= TC_SEQ_HANDLER_EVAL;
			ELSE
				CASE Internal.CurrentWait OF
					TC_SEQ_WAIT_FALSE:
						IF Internal.CTON_0.Q THEN
							Out.Status.Timeout				:= TRUE;
							Internal.State					:= TC_SEQ_HANDLER_INTERRUPT;
						END_IF;
					TC_SEQ_WAIT_TRUE:
						Internal.State						:= TC_SEQ_HANDLER_EVAL;
					TC_SEQ_WAIT_INTERRUPT:
						Out.Status.Interrupt				:= TRUE;
						Internal.State						:= TC_SEQ_HANDLER_INTERRUPT;
					TC_SEQ_WAIT_ERROR:
						Out.Status.Processing				:= FALSE;
						Out.Status.Error					:= TRUE;
						Internal.ErrorID.30					:= 1;
						Internal.State						:= TC_SEQ_HANDLER_ERROR;
					ELSE
						Out.Status.Processing				:= FALSE;
						Out.Status.Error					:= TRUE;
						Internal.ErrorID.29					:= 1;
						Internal.State						:= TC_SEQ_HANDLER_ERROR;
				END_CASE;
			END_IF
		TC_SEQ_HANDLER_DELAY:
			Out.Status.CurrentState						:= 'TC_SEQ_HANDLER_DELAY';
			Out.Status.Processing						:= TRUE;
			Internal.CTON_0.IN							:= TRUE;
			Internal.CTON_0.PT							:= LREAL_TO_TIME(Internal.CurrentDelay*1000.0);
			Internal.CTON_0.PAUSE						:= FALSE;
			IF ForceNext = TRUE THEN
				Internal.State							:= TC_SEQ_HANDLER_EVAL;
			ELSIF Internal.CTON_0.Q OR Internal.CurrentDelay = 0 THEN
				Internal.State							:= TC_SEQ_HANDLER_EVAL;
			END_IF;
		TC_SEQ_HANDLER_INTERRUPT:
			Out.Status.CurrentState						:= 'TC_SEQ_HANDLER_INTERRUPT';
			Out.Status.Processing						:= TRUE;
			IF ForceNext = TRUE THEN
				Internal.State							:= TC_SEQ_HANDLER_EVAL;
			ELSIF Pause THEN
				Out.Status.Processing					:= FALSE;
				Out.Status.Paused						:= TRUE;
			ELSIF ClearBuffer THEN
				Internal.State							:= TC_SEQ_HANDLER_EVAL;
			ELSE
				Out.Status.Processing					:= FALSE;
				Out.Status.Error						:= TRUE;
				Internal.ErrorID.31						:= 1;
				Internal.State							:= TC_SEQ_HANDLER_ERROR;
			END_IF
		TC_SEQ_HANDLER_ERROR:
			Out.Status.CurrentState						:= 'TC_SEQ_HANDLER_ERROR';
			Out.Status.Error							:= TRUE;
			IF ErrorReset THEN
				Internal.State							:= TC_SEQ_HANDLER_RESET;
			END_IF;
	END_CASE;
	IF Internal.LastState <> Internal.State THEN
		Internal.LastState 								:= Internal.State;
		Internal.CTON_0(IN := FALSE, PT := T#0ms, PAUSE := FALSE);
	ELSE
		Internal.CTON_0();
		Out.Status.Elapsed								:= TIME_TO_LREAL(Internal.CTON_0.ET)/1000.0;
		Out.Status.Remaining							:= TIME_TO_LREAL(Internal.CTON_0.PT)/1000.0 - Out.Status.Elapsed;
	END_IF;
	IF brsmemcmp(ADR(Out.Buffer.Current),ADR(Internal.CurrentBuffer),SIZEOF(Internal.CurrentBuffer)) <> 0 AND Internal.CurrentBuffer.Type <> TC_SEQ_TYPE_NONE THEN
		IF MAX_TC_SEQ_BUFFER_LAST_IDX > 0 THEN
			brsmemmove(ADR(Out.Buffer.Last[1]),ADR(Out.Buffer.Last[0]),SIZEOF(Out.Buffer.Last)-SIZEOF(Out.Buffer.Last[0]));
		END_IF;
		brsmemcpy(ADR(Out.Buffer.Last[0]),ADR(Internal.CurrentBuffer),SIZEOF(Internal.CurrentBuffer));
	END_IF;
	brsmemcpy(ADR(Out.Buffer.Current),ADR(Internal.CurrentBuffer),SIZEOF(Internal.CurrentBuffer));
	Out.Status.ErrorID									:= Internal.ErrorID;
END_FUNCTION_BLOCK
```

#### TC_Seq_EnumStringSearch.st
```iecst
(* Finds the index of the enum string *)
FUNCTION TC_Seq_EnumStringSearch
	TC_Seq_EnumStringSearch := -1;
	brsmemset(ADR(Internal),0,SIZEOF(Internal));
	IF EnumNameSTRING <> '' AND EnumValueSTRING <> '' THEN
		TC_brsstrcat(ADR(Internal.PvRoot),ADR('gES.'),SIZEOF(Internal.PvRoot));
		TC_brsstrcat(ADR(Internal.PvRoot),ADR(EnumNameSTRING),SIZEOF(Internal.PvRoot));
		Internal.Status := PV_ninfo(ADR(Internal.PvRoot),ADR(Internal.Datatype),ADR(Internal.DataLen),ADR(Internal.Dimension));
		IF Internal.Status = 0 AND Internal.Dimension > 0 THEN
			FOR Internal.i := 0 TO UINT_TO_DINT(Internal.Dimension-1) DO
				Internal.IdxString := DINT_TO_STRING(Internal.i);
				brsmemset(ADR(Internal.PvName),0,SIZEOF(Internal.PvName));
				TC_brsstrcat(ADR(Internal.PvName),ADR(Internal.PvRoot),SIZEOF(Internal.PvName));
				TC_brsstrcat(ADR(Internal.PvName),ADR('['),SIZEOF(Internal.PvName));
				TC_brsstrcat(ADR(Internal.PvName),ADR(Internal.IdxString),SIZEOF(Internal.PvName));
				TC_brsstrcat(ADR(Internal.PvName),ADR(']'),SIZEOF(Internal.PvName));
				Internal.Status := PV_xgetadr(ADR(Internal.PvName),ADR(Internal.PvAddress),ADR(Internal.PvLen));
				IF Internal.Status = 0 AND SIZEOF(Internal.PvValue) = Internal.PvLen THEN
					brsmemcpy(ADR(Internal.PvValue),Internal.PvAddress,SIZEOF(Internal.PvValue)-1);
					IF EnumValueSTRING = Internal.PvValue THEN
						TC_Seq_EnumStringSearch := Internal.i;
						EXIT;
					END_IF;
				ELSE
					EXIT;
				END_IF;
			END_FOR;
		END_IF;
	END_IF;
END_FUNCTION
```

#### TC_Seq_JsonToElem.st
```iecst
FUNCTION TC_Seq_JsonToElem
	brsmemset(ADR(Internal),0,SIZEOF(Internal));
	TC_Seq_JsonToElem := 0;
	IF pJsonString = 0 OR pElement = 0 THEN
		TC_Seq_JsonToElem.0 := TRUE;
		RETURN;
	END_IF;
	brsmemset(pElement,0,SIZEOF(Internal.Element));
	Internal.TC_JSON_Parse_0(Enable := TRUE, pBuffer := pJsonString, pPairs := ADR(Internal.JSONPairs), NoQuotes := TRUE);
	IF Internal.TC_JSON_Parse_0.Error THEN
		TC_Seq_JsonToElem.1 := TRUE;
		RETURN;
	END_IF;
	Internal.TC_JSON_Parse_0(Enable := FALSE);
	FOR Internal.i := 0 TO MAX_JSON_PARSE_PAIR_IDX DO
		IF Internal.JSONPairs[Internal.i].Name = '' AND Internal.JSONPairs[Internal.i].Value = '' THEN
			EXIT;
		ELSE
			IF Internal.JSONPairs[Internal.i].Name = 'par' THEN
				IF Internal.Par = '' THEN
					TC_brsstrcat(ADR(Internal.Par),ADR('{'),SIZEOF(Internal.Par));
				ELSE
					Internal.ParDone := TRUE;
					TC_brsstrcat(ADR(Internal.Par),ADR('}'),SIZEOF(Internal.Par));
				END_IF;
			ELSIF NOT Internal.ParDone AND Internal.Par <> '' THEN
				IF Internal.Par <> '{' THEN
					TC_brsstrcat(ADR(Internal.Par),ADR(','),SIZEOF(Internal.Par));
				END_IF;
				TC_brsstrcat(ADR(Internal.Par),ADR('"'),SIZEOF(Internal.Par));
				TC_brsstrcat(ADR(Internal.Par),ADR(Internal.JSONPairs[Internal.i].Name),SIZEOF(Internal.Par));
				TC_brsstrcat(ADR(Internal.Par),ADR('":"'),SIZEOF(Internal.Par));
				TC_brsstrcat(ADR(Internal.Par),ADR(Internal.JSONPairs[Internal.i].Value),SIZEOF(Internal.Par));
				TC_brsstrcat(ADR(Internal.Par),ADR('"'),SIZEOF(Internal.Par));
			ELSIF Internal.JSONPairs[Internal.i].Name = 'type' THEN
				IF Internal.JSONPairs[Internal.i].Value = 'D' THEN
					Internal.Element.Type 	:= TC_SEQ_TYPE_DELAY;
				ELSIF Internal.JSONPairs[Internal.i].Value = 'W' THEN
					Internal.Element.Type 	:= TC_SEQ_TYPE_WAIT;
				ELSIF Internal.JSONPairs[Internal.i].Value = 'C' THEN
					Internal.Element.Type 	:= TC_SEQ_TYPE_CMD;
				ELSIF Internal.JSONPairs[Internal.i].Value = 'M' THEN
					Internal.Element.Type 	:= TC_SEQ_TYPE_MON;
				ELSE
					TC_Seq_JsonToElem.2 	:= TRUE;
					RETURN;
				END_IF;
			ELSIF Internal.JSONPairs[Internal.i].Name = 'driver' THEN
				Internal.Driver 	:= Internal.JSONPairs[Internal.i].Value;
			ELSIF Internal.JSONPairs[Internal.i].Name = 'ident' THEN
				Internal.Ident 		:= Internal.JSONPairs[Internal.i].Value;
			ELSIF Internal.JSONPairs[Internal.i].Name = 'inst' THEN
				Internal.Inst 		:= Internal.JSONPairs[Internal.i].Value;
			ELSIF Internal.JSONPairs[Internal.i].Name = 'time' THEN
				Internal.Element.Time 		:= STRING_TO_LREAL(Internal.JSONPairs[Internal.i].Value);
			ELSIF Internal.JSONPairs[Internal.i].Name = 'enable' THEN
				Internal.Enable 	:= STRING_TO_BOOL(Internal.JSONPairs[Internal.i].Value);
			ELSIF Internal.JSONPairs[Internal.i].Name = 'sev' THEN
				Internal.Sev 		:= STRING_TO_DINT(Internal.JSONPairs[Internal.i].Value);
			END_IF;
		END_IF;
	END_FOR;

	IF Internal.Element.Type = TC_SEQ_TYPE_DELAY THEN
		brsmemcpy(pElement,ADR(Internal.Element),SIZEOF(Internal.Element));
		RETURN;
	ELSIF Internal.Driver = '' OR Internal.Inst = '' OR Internal.Ident = '' THEN
		TC_Seq_JsonToElem.3 := TRUE;
		brsmemset(pElement,0,SIZEOF(Internal.Element));
		RETURN;
	END_IF;

	TC_brsstrcat(ADR(Internal.EnumNameString_Inst),ADR('DRIVER_INST_'),SIZEOF(Internal.EnumNameString_Inst));
	TC_brsstrcat(ADR(Internal.EnumNameString_Inst),ADR(Internal.Driver),SIZEOF(Internal.EnumNameString_Inst));
	TC_brsstrcat(ADR(Internal.EnumNameString_Inst),ADR('_ENUM'),SIZEOF(Internal.EnumNameString_Inst));
	TC_brsstrcat(ADR(Internal.EnumValueString_Inst),ADR('DRIVER_INST_'),SIZEOF(Internal.EnumValueString_Inst));
	TC_brsstrcat(ADR(Internal.EnumValueString_Inst),ADR(Internal.Driver),SIZEOF(Internal.EnumValueString_Inst));
	TC_brsstrcat(ADR(Internal.EnumValueString_Inst),ADR('_'),SIZEOF(Internal.EnumValueString_Inst));
	TC_brsstrcat(ADR(Internal.EnumValueString_Inst),ADR(Internal.Inst),SIZEOF(Internal.EnumValueString_Inst));
	Internal.InstIdx := TC_Seq_EnumStringSearch(Internal.EnumNameString_Inst,Internal.EnumValueString_Inst);
	IF Internal.InstIdx < 0 THEN
		TC_Seq_JsonToElem.4 := TRUE;
		brsmemset(pElement,0,SIZEOF(Internal.Element));
		RETURN;
	END_IF;

	IF Internal.Element.Type = TC_SEQ_TYPE_WAIT THEN
		TC_brsstrcat(ADR(Internal.EnumNameString_Ident),ADR('W_'),SIZEOF(Internal.EnumNameString_Ident));
		TC_brsstrcat(ADR(Internal.EnumNameString_Ident),ADR(Internal.Driver),SIZEOF(Internal.EnumNameString_Ident));
		TC_brsstrcat(ADR(Internal.EnumNameString_Ident),ADR('_ENUM'),SIZEOF(Internal.EnumNameString_Ident));
		TC_brsstrcat(ADR(Internal.EnumValueString_Ident),ADR('W_'),SIZEOF(Internal.EnumValueString_Ident));
		TC_brsstrcat(ADR(Internal.EnumValueString_Ident),ADR(Internal.Driver),SIZEOF(Internal.EnumValueString_Ident));
		TC_brsstrcat(ADR(Internal.EnumValueString_Ident),ADR('_'),SIZEOF(Internal.EnumValueString_Ident));
		TC_brsstrcat(ADR(Internal.EnumValueString_Ident),ADR(Internal.Ident),SIZEOF(Internal.EnumValueString_Ident));
		Internal.IdentIdx := TC_Seq_EnumStringSearch(Internal.EnumNameString_Ident,Internal.EnumValueString_Ident);
		IF Internal.IdentIdx < 0 THEN
			TC_Seq_JsonToElem.5 := TRUE;
			brsmemset(pElement,0,SIZEOF(Internal.Element));
			RETURN;
		END_IF;
		brsmemset(ADR(Internal.PvName),0,SIZEOF(Internal.PvName));
		TC_brsstrcat(ADR(Internal.PvName),ADR('gDriver.'),SIZEOF(Internal.PvName));
		TC_brsstrcat(ADR(Internal.PvName),ADR(Internal.Driver),SIZEOF(Internal.PvName));
		TC_brsstrcat(ADR(Internal.PvName),ADR('['),SIZEOF(Internal.PvName));
		Internal.InstIdxString := DINT_TO_STRING(Internal.InstIdx);
		TC_brsstrcat(ADR(Internal.PvName),ADR(Internal.InstIdxString),SIZEOF(Internal.PvName));
		TC_brsstrcat(ADR(Internal.PvName),ADR('].Wait['),SIZEOF(Internal.PvName));
		Internal.IdentIdxString := DINT_TO_STRING(Internal.IdentIdx);
		TC_brsstrcat(ADR(Internal.PvName),ADR(Internal.IdentIdxString),SIZEOF(Internal.PvName));
		TC_brsstrcat(ADR(Internal.PvName),ADR(']'),SIZEOF(Internal.PvName));
		Internal.Status := PV_xgetadr(ADR(Internal.PvName),ADR(Internal.PvAddress),ADR(Internal.PvLen));
		IF Internal.Status = 0 AND Internal.PvLen = 4 THEN
			Internal.WaitPvAddress := Internal.PvAddress;
			Internal.Element.WaitPvAddress := Internal.PvAddress;
			brsmemcpy(ADR(Internal.Element.Json),pJsonString,SIZEOF(Internal.Element.Json));
			brsmemcpy(pElement,ADR(Internal.Element),SIZEOF(Internal.Element));
		ELSE
			TC_Seq_JsonToElem.6 		:= TRUE;
			brsmemset(pElement,0,SIZEOF(Internal.Element));
			RETURN;
		END_IF;
	ELSIF Internal.Element.Type = TC_SEQ_TYPE_MON THEN
		TC_brsstrcat(ADR(Internal.EnumNameString_Ident),ADR('M_'),SIZEOF(Internal.EnumNameString_Ident));
		TC_brsstrcat(ADR(Internal.EnumNameString_Ident),ADR(Internal.Driver),SIZEOF(Internal.EnumNameString_Ident));
		TC_brsstrcat(ADR(Internal.EnumNameString_Ident),ADR('_ENUM'),SIZEOF(Internal.EnumNameString_Ident));
		TC_brsstrcat(ADR(Internal.EnumValueString_Ident),ADR('M_'),SIZEOF(Internal.EnumValueString_Ident));
		TC_brsstrcat(ADR(Internal.EnumValueString_Ident),ADR(Internal.Driver),SIZEOF(Internal.EnumValueString_Ident));
		TC_brsstrcat(ADR(Internal.EnumValueString_Ident),ADR('_'),SIZEOF(Internal.EnumValueString_Ident));
		TC_brsstrcat(ADR(Internal.EnumValueString_Ident),ADR(Internal.Ident),SIZEOF(Internal.EnumValueString_Ident));
		Internal.IdentIdx := TC_Seq_EnumStringSearch(Internal.EnumNameString_Ident,Internal.EnumValueString_Ident);
		IF Internal.IdentIdx < 0 THEN
			TC_Seq_JsonToElem.7 := TRUE;
			brsmemset(pElement,0,SIZEOF(Internal.Element));
			RETURN;
		END_IF;
		brsmemset(ADR(Internal.PvName),0,SIZEOF(Internal.PvName));
		TC_brsstrcat(ADR(Internal.PvName),ADR('gDriver.'),SIZEOF(Internal.PvName));
		TC_brsstrcat(ADR(Internal.PvName),ADR(Internal.Driver),SIZEOF(Internal.PvName));
		TC_brsstrcat(ADR(Internal.PvName),ADR('['),SIZEOF(Internal.PvName));
		Internal.InstIdxString := DINT_TO_STRING(Internal.InstIdx);
		TC_brsstrcat(ADR(Internal.PvName),ADR(Internal.InstIdxString),SIZEOF(Internal.PvName));
		TC_brsstrcat(ADR(Internal.PvName),ADR('].Par.Mon['),SIZEOF(Internal.PvName));
		Internal.IdentIdxString := DINT_TO_STRING(Internal.IdentIdx);
		TC_brsstrcat(ADR(Internal.PvName),ADR(Internal.IdentIdxString),SIZEOF(Internal.PvName));
		TC_brsstrcat(ADR(Internal.PvName),ADR(']'),SIZEOF(Internal.PvName));
		brsmemset(ADR(Internal.PvNameSub),0,SIZEOF(Internal.PvNameSub));
		TC_brsstrcat(ADR(Internal.PvNameSub),ADR(Internal.PvName),SIZEOF(Internal.PvNameSub));
		TC_brsstrcat(ADR(Internal.PvNameSub),ADR('.Enable'),SIZEOF(Internal.PvNameSub));
		Internal.Status := PV_xgetadr(ADR(Internal.PvNameSub),ADR(Internal.PvAddress),ADR(Internal.PvLen));
		IF Internal.Status = 0 AND Internal.PvLen = 1 THEN
			brsmemcpy(Internal.PvAddress,ADR(Internal.Enable),SIZEOF(Internal.Enable));
		ELSE
			TC_Seq_JsonToElem.8 		:= TRUE;
			brsmemset(pElement,0,SIZEOF(Internal.Element));
			RETURN;
		END_IF;
		brsmemset(ADR(Internal.PvNameSub),0,SIZEOF(Internal.PvNameSub));
		TC_brsstrcat(ADR(Internal.PvNameSub),ADR(Internal.PvName),SIZEOF(Internal.PvNameSub));
		TC_brsstrcat(ADR(Internal.PvNameSub),ADR('.Sev'),SIZEOF(Internal.PvNameSub));
		Internal.Status := PV_xgetadr(ADR(Internal.PvNameSub),ADR(Internal.PvAddress),ADR(Internal.PvLen));
		IF Internal.Status = 0 AND Internal.PvLen = 4 THEN
			brsmemcpy(Internal.PvAddress,ADR(Internal.Sev),SIZEOF(Internal.Sev));
		ELSE
			TC_Seq_JsonToElem.9 		:= TRUE;
			brsmemset(pElement,0,SIZEOF(Internal.Element));
			RETURN;
		END_IF;
		brsmemset(ADR(Internal.PvNameSub),0,SIZEOF(Internal.PvNameSub));
		TC_brsstrcat(ADR(Internal.PvNameSub),ADR(Internal.PvName),SIZEOF(Internal.PvNameSub));
		TC_brsstrcat(ADR(Internal.PvNameSub),ADR('.Time'),SIZEOF(Internal.PvNameSub));
		Internal.Status := PV_xgetadr(ADR(Internal.PvNameSub),ADR(Internal.PvAddress),ADR(Internal.PvLen));
		IF Internal.Status = 0 AND Internal.PvLen = 8 THEN
			brsmemcpy(Internal.PvAddress,ADR(Internal.Element.Time),SIZEOF(Internal.Element.Time));
		ELSE
			TC_Seq_JsonToElem.10 		:= TRUE;
			brsmemset(pElement,0,SIZEOF(Internal.Element));
			RETURN;
		END_IF;
		brsmemcpy(ADR(Internal.Element.Json),pJsonString,SIZEOF(Internal.Element.Json));
		brsmemcpy(pElement,ADR(Internal.Element),SIZEOF(Internal.Element));
	ELSIF Internal.Element.Type = TC_SEQ_TYPE_CMD THEN
		TC_brsstrcat(ADR(Internal.EnumNameString_Ident),ADR('C_'),SIZEOF(Internal.EnumNameString_Ident));
		TC_brsstrcat(ADR(Internal.EnumNameString_Ident),ADR(Internal.Driver),SIZEOF(Internal.EnumNameString_Ident));
		TC_brsstrcat(ADR(Internal.EnumNameString_Ident),ADR('_ENUM'),SIZEOF(Internal.EnumNameString_Ident));
		TC_brsstrcat(ADR(Internal.EnumValueString_Ident),ADR('C_'),SIZEOF(Internal.EnumValueString_Ident));
		TC_brsstrcat(ADR(Internal.EnumValueString_Ident),ADR(Internal.Driver),SIZEOF(Internal.EnumValueString_Ident));
		TC_brsstrcat(ADR(Internal.EnumValueString_Ident),ADR('_'),SIZEOF(Internal.EnumValueString_Ident));
		TC_brsstrcat(ADR(Internal.EnumValueString_Ident),ADR(Internal.Ident),SIZEOF(Internal.EnumValueString_Ident));
		Internal.IdentIdx := TC_Seq_EnumStringSearch(Internal.EnumNameString_Ident,Internal.EnumValueString_Ident);
		IF Internal.IdentIdx < 0 THEN
			TC_Seq_JsonToElem.11 := TRUE;
			brsmemset(pElement,0,SIZEOF(Internal.Element));
			RETURN;
		END_IF;
		brsmemset(ADR(Internal.PvName),0,SIZEOF(Internal.PvName));
		TC_brsstrcat(ADR(Internal.DriverRoot),ADR('gDriver.'),SIZEOF(Internal.DriverRoot));
		TC_brsstrcat(ADR(Internal.DriverRoot),ADR(Internal.Driver),SIZEOF(Internal.DriverRoot));
		TC_brsstrcat(ADR(Internal.DriverRoot),ADR('['),SIZEOF(Internal.DriverRoot));
		Internal.InstIdxString := DINT_TO_STRING(Internal.InstIdx);
		TC_brsstrcat(ADR(Internal.DriverRoot),ADR(Internal.InstIdxString),SIZEOF(Internal.DriverRoot));
		TC_brsstrcat(ADR(Internal.DriverRoot),ADR('].'),SIZEOF(Internal.DriverRoot));
		TC_brsstrcat(ADR(Internal.PvName),ADR(Internal.DriverRoot),SIZEOF(Internal.PvName));
		TC_brsstrcat(ADR(Internal.PvName),ADR('Cmd['),SIZEOF(Internal.PvName));
		Internal.IdentIdxString := DINT_TO_STRING(Internal.IdentIdx);
		TC_brsstrcat(ADR(Internal.PvName),ADR(Internal.IdentIdxString),SIZEOF(Internal.PvName));
		TC_brsstrcat(ADR(Internal.PvName),ADR(']'),SIZEOF(Internal.PvName));
		Internal.Status := PV_xgetadr(ADR(Internal.PvName),ADR(Internal.PvAddress),ADR(Internal.PvLen));
		IF Internal.Status = 0 AND Internal.PvLen = 1 THEN
			Internal.CmdPvAddress := Internal.PvAddress;
		ELSE
			TC_Seq_JsonToElem.12 		:= TRUE;
			brsmemset(pElement,0,SIZEOF(Internal.Element));
			RETURN;
		END_IF;

		brsmemset(ADR(Internal.JSONPairs),0,SIZEOF(Internal.JSONPairs));
		Internal.TC_JSON_Parse_0(Enable := TRUE, pBuffer := ADR(Internal.Par), pPairs := ADR(Internal.JSONPairs), NoQuotes := TRUE);
		IF Internal.TC_JSON_Parse_0.Error THEN
			TC_Seq_JsonToElem.13 := TRUE;
			brsmemset(pElement,0,SIZEOF(Internal.Element));
			RETURN;
		END_IF;
		Internal.TC_JSON_Parse_0(Enable := FALSE);
		Internal.idx := 0;
		FOR Internal.i := 0 TO MAX_JSON_PARSE_PAIR_IDX DO
			IF Internal.JSONPairs[Internal.i].Name = '' AND Internal.JSONPairs[Internal.i].Value = '' THEN
				EXIT;
			ELSIF Internal.JSONPairs[Internal.i].Name <> '' THEN
				brsmemset(ADR(Internal.ParDataType),0,SIZEOF(Internal.ParDataType));
				brsmemcpy(ADR(Internal.ParDataType),ADR(Internal.JSONPairs[Internal.i].Value)+1,2);
				brsmemset(ADR(Internal.ParValue),0,SIZEOF(Internal.ParValue));
				brsmemcpy(ADR(Internal.ParValue),ADR(Internal.JSONPairs[Internal.i].Value)+4,MAX_JSON_PARSE_VALUE_LEN-4);
				brsmemset(ADR(Internal.PvName),0,SIZEOF(Internal.PvName));
				TC_brsstrcat(ADR(Internal.PvName),ADR(Internal.DriverRoot),SIZEOF(Internal.PvName));
				TC_brsstrcat(ADR(Internal.PvName),ADR('Par.'),SIZEOF(Internal.PvName));
				TC_brsstrcat(ADR(Internal.PvName),ADR(Internal.JSONPairs[Internal.i].Name),SIZEOF(Internal.PvName));
				Internal.ParElement[Internal.idx].Name := Internal.PvName;
				Internal.Status := PV_ninfo(ADR(Internal.PvName),ADR(Internal.Datatype),ADR(Internal.DataLen),ADR(Internal.Dimension));
				IF Internal.Status <> 0 THEN
					TC_Seq_JsonToElem.14 := TRUE;
					brsmemset(pElement,0,SIZEOF(Internal.Element));
					RETURN;
				END_IF;
				IF Internal.Datatype = SYSLIB_IEC_TYPE_BOOL AND Internal.ParDataType = 'BO' THEN
					Internal.ParElement[Internal.idx].GenVar.Select 			:= TC_SEQ_PAR_SELECT_BOOL;
					Internal.ParElement[Internal.idx].GenVar.VarBOOL 			:= STRING_TO_BOOL(Internal.ParValue);
				ELSIF Internal.Datatype = SYSLIB_IEC_TYPE_SINT AND Internal.ParDataType = 'SS' THEN
					Internal.ParElement[Internal.idx].GenVar.Select 			:= TC_SEQ_PAR_SELECT_SINT;
					Internal.ParElement[Internal.idx].GenVar.VarSINT 			:= STRING_TO_SINT(Internal.ParValue);
				ELSIF Internal.Datatype = SYSLIB_IEC_TYPE_USINT AND Internal.ParDataType = 'US' THEN
					Internal.ParElement[Internal.idx].GenVar.Select 			:= TC_SEQ_PAR_SELECT_USINT;
					Internal.ParElement[Internal.idx].GenVar.VarUSINT 		:= STRING_TO_USINT(Internal.ParValue);
				ELSIF Internal.Datatype = SYSLIB_IEC_TYPE_INT AND Internal.ParDataType = 'SI' THEN
					Internal.ParElement[Internal.idx].GenVar.Select 			:= TC_SEQ_PAR_SELECT_INT;
					Internal.ParElement[Internal.idx].GenVar.VarINT 			:= STRING_TO_INT(Internal.ParValue);
				ELSIF Internal.Datatype = SYSLIB_IEC_TYPE_UINT AND Internal.ParDataType = 'UI' THEN
					Internal.ParElement[Internal.idx].GenVar.Select 			:= TC_SEQ_PAR_SELECT_UINT;
					Internal.ParElement[Internal.idx].GenVar.VarUINT 			:= STRING_TO_UINT(Internal.ParValue);
				ELSIF (Internal.Datatype = SYSLIB_IEC_TYPE_DINT OR Internal.Datatype = SYSLIB_IEC_TYPE_USER_DEFINED) AND Internal.ParDataType = 'SD' THEN
					Internal.ParElement[Internal.idx].GenVar.Select 			:= TC_SEQ_PAR_SELECT_DINT;
					Internal.ParElement[Internal.idx].GenVar.VarDINT 			:= STRING_TO_DINT(Internal.ParValue);
				ELSIF Internal.Datatype = SYSLIB_IEC_TYPE_UDINT AND Internal.ParDataType = 'UD' THEN
					Internal.ParElement[Internal.idx].GenVar.Select 			:= TC_SEQ_PAR_SELECT_UDINT;
					Internal.ParElement[Internal.idx].GenVar.VarUDINT 		:= STRING_TO_UDINT(Internal.ParValue);
				ELSIF Internal.Datatype = SYSLIB_IEC_TYPE_REAL AND Internal.ParDataType = 'RR' THEN
					Internal.ParElement[Internal.idx].GenVar.Select 			:= TC_SEQ_PAR_SELECT_REAL;
					Internal.ParElement[Internal.idx].GenVar.VarREAL 			:= STRING_TO_REAL(Internal.ParValue);
				ELSIF Internal.Datatype = SYSLIB_IEC_TYPE_LREAL AND Internal.ParDataType = 'LR' THEN
					Internal.ParElement[Internal.idx].GenVar.Select 			:= TC_SEQ_PAR_SELECT_LREAL;
					Internal.ParElement[Internal.idx].GenVar.VarLREAL 		:= STRING_TO_LREAL(Internal.ParValue);
				ELSIF Internal.Datatype = SYSLIB_IEC_TYPE_TIME AND Internal.ParDataType = 'TM' THEN
					Internal.ParElement[Internal.idx].GenVar.Select 			:= TC_SEQ_PAR_SELECT_TIME;
					Internal.ParElement[Internal.idx].GenVar.VarTIME 			:= STRING_TO_TIME(Internal.ParValue);
				ELSIF Internal.Datatype = SYSLIB_IEC_TYPE_DATE_AND_TIME AND Internal.ParDataType = 'DT' THEN
					Internal.ParElement[Internal.idx].GenVar.Select 			:= TC_SEQ_PAR_SELECT_DT;
					Internal.ParElement[Internal.idx].GenVar.VarDT 			:= STRING_TO_DT(Internal.ParValue);
				ELSIF Internal.Datatype = SYSLIB_IEC_TYPE_STRING AND Internal.ParDataType = 'ST' THEN
					Internal.ParElement[Internal.idx].GenVar.Select 			:= TC_SEQ_PAR_SELECT_STRING;
					Internal.ParElement[Internal.idx].GenVar.VarSTRING 		:= Internal.ParValue;
				ELSIF Internal.Datatype = SYSLIB_IEC_TYPE_UDINT AND Internal.ParDataType = 'SA' THEN
					Internal.ParElement[Internal.idx].GenVar.Select 			:= TC_SEQ_PAR_SELECT_STRINGADR;
					Internal.ParElement[Internal.idx].GenVar.VarSTRING_ADR 	:= STRING_TO_UDINT(Internal.ParValue);
				ELSIF Internal.Datatype = SYSLIB_IEC_TYPE_UDINT AND Internal.ParDataType = 'AD' THEN
					Internal.ParElement[Internal.idx].GenVar.Select 			:= TC_SEQ_PAR_SELECT_ADR;
					Internal.ParElement[Internal.idx].GenVar.VarADR 			:= STRING_TO_UDINT(Internal.ParValue);
				ELSIF Internal.Datatype = SYSLIB_IEC_TYPE_UDINT AND Internal.ParDataType = 'PR' THEN
					Internal.ParElement[Internal.idx].GenVar.Select 			:= TC_SEQ_PAR_SELECT_PTR;
					Internal.ParElement[Internal.idx].GenVar.VarADR 			:= STRING_TO_UDINT(Internal.ParValue);//TODO: How to assign access a pointer instead of a value...
				ELSIF Internal.Datatype = SYSLIB_IEC_TYPE_DINT AND Internal.ParDataType = 'EN' THEN
					Internal.ParElement[Internal.idx].GenVar.Select 			:= TC_SEQ_PAR_SELECT_ENUMNAME;
					Internal.ParElement[Internal.idx].GenVar.VarENUM 			:= STRING_TO_DINT(Internal.ParValue);//TODO: Use gES? How to get the enum name to value...
					Internal.ParElement[Internal.idx].GenVar.VarENUM_STRING	:= Internal.ParValue;
				ELSE
					TC_Seq_JsonToElem.15 := TRUE;
					brsmemset(pElement,0,SIZEOF(Internal.Element));
					RETURN;
				END_IF;
				Internal.idx := Internal.idx + 1;
			END_IF;
		END_FOR;

		FOR Internal.i := 0 TO MAX_JSON_PARSE_PAIR_IDX DO
			IF Internal.ParElement[Internal.i].GenVar.Select = TC_SEQ_PAR_SELECT_NULL THEN
				EXIT;
			ELSE
				Internal.Status := PV_xgetadr(ADR(Internal.ParElement[Internal.i].Name),ADR(Internal.PvAddress),ADR(Internal.PvLen));
				IF Internal.Status <> 0 THEN
					TC_Seq_JsonToElem.16 		:= TRUE;
					brsmemset(pElement,0,SIZEOF(Internal.Element));
					RETURN;
				END_IF;
				CASE Internal.ParElement[Internal.i].GenVar.Select OF
					TC_SEQ_PAR_SELECT_BOOL:
						brsmemcpy(Internal.PvAddress,ADR(Internal.ParElement[Internal.i].GenVar.VarBOOL),SIZEOF(Internal.ParElement[Internal.i].GenVar.VarBOOL));
					TC_SEQ_PAR_SELECT_INT:
						brsmemcpy(Internal.PvAddress,ADR(Internal.ParElement[Internal.i].GenVar.VarINT),SIZEOF(Internal.ParElement[Internal.i].GenVar.VarINT));
					TC_SEQ_PAR_SELECT_USINT:
						brsmemcpy(Internal.PvAddress,ADR(Internal.ParElement[Internal.i].GenVar.VarUSINT),SIZEOF(Internal.ParElement[Internal.i].GenVar.VarUSINT));
					TC_SEQ_PAR_SELECT_SINT:
						brsmemcpy(Internal.PvAddress,ADR(Internal.ParElement[Internal.i].GenVar.VarSINT),SIZEOF(Internal.ParElement[Internal.i].GenVar.VarSINT));
					TC_SEQ_PAR_SELECT_UINT:
						brsmemcpy(Internal.PvAddress,ADR(Internal.ParElement[Internal.i].GenVar.VarUINT),SIZEOF(Internal.ParElement[Internal.i].GenVar.VarUINT));
					TC_SEQ_PAR_SELECT_DINT:
						brsmemcpy(Internal.PvAddress,ADR(Internal.ParElement[Internal.i].GenVar.VarDINT),SIZEOF(Internal.ParElement[Internal.i].GenVar.VarDINT));
					TC_SEQ_PAR_SELECT_UDINT:
						brsmemcpy(Internal.PvAddress,ADR(Internal.ParElement[Internal.i].GenVar.VarUDINT),SIZEOF(Internal.ParElement[Internal.i].GenVar.VarUDINT));
					TC_SEQ_PAR_SELECT_REAL:
						brsmemcpy(Internal.PvAddress,ADR(Internal.ParElement[Internal.i].GenVar.VarREAL),SIZEOF(Internal.ParElement[Internal.i].GenVar.VarREAL));
					TC_SEQ_PAR_SELECT_LREAL:
						brsmemcpy(Internal.PvAddress,ADR(Internal.ParElement[Internal.i].GenVar.VarLREAL),SIZEOF(Internal.ParElement[Internal.i].GenVar.VarLREAL));
					TC_SEQ_PAR_SELECT_TIME:
						brsmemcpy(Internal.PvAddress,ADR(Internal.ParElement[Internal.i].GenVar.VarTIME),SIZEOF(Internal.ParElement[Internal.i].GenVar.VarTIME));
					TC_SEQ_PAR_SELECT_DT:
						brsmemcpy(Internal.PvAddress,ADR(Internal.ParElement[Internal.i].GenVar.VarDT),SIZEOF(Internal.ParElement[Internal.i].GenVar.VarDT));
					TC_SEQ_PAR_SELECT_ENUMNAME:
						brsmemcpy(Internal.PvAddress,ADR(Internal.ParElement[Internal.i].GenVar.VarENUM),SIZEOF(Internal.ParElement[Internal.i].GenVar.VarENUM));
					TC_SEQ_PAR_SELECT_STRING:
						IF Internal.PvLen <= brsstrlen(ADR(Internal.ParElement[Internal.i].GenVar.VarSTRING)) THEN
							TC_Seq_JsonToElem.17 		:= TRUE;
							brsmemset(pElement,0,SIZEOF(Internal.Element));
							RETURN;
						END_IF;
						brsmemset(Internal.PvAddress,0,Internal.PvLen);
						brsmemcpy(Internal.PvAddress,ADR(Internal.ParElement[Internal.i].GenVar.VarSTRING),brsstrlen(ADR(Internal.ParElement[Internal.i].GenVar.VarSTRING)));
					TC_SEQ_PAR_SELECT_STRINGADR:
						IF Internal.PvLen <= brsstrlen(Internal.ParElement[Internal.i].GenVar.VarSTRING_ADR) THEN
							TC_Seq_JsonToElem.18 		:= TRUE;
							brsmemset(pElement,0,SIZEOF(Internal.Element));
							RETURN;
						END_IF;
						brsmemset(Internal.PvAddress,0,Internal.PvLen);
						brsmemcpy(Internal.PvAddress,Internal.ParElement[Internal.i].GenVar.VarSTRING_ADR,brsstrlen(Internal.ParElement[Internal.i].GenVar.VarSTRING_ADR));
					TC_SEQ_PAR_SELECT_ADR:
						brsmemcpy(Internal.PvAddress,ADR(Internal.ParElement[Internal.i].GenVar.VarADR),SIZEOF(Internal.ParElement[Internal.i].GenVar.VarADR));
					TC_SEQ_PAR_SELECT_PTR:
						brsmemcpy(Internal.PvAddress,ADR(Internal.ParElement[Internal.i].GenVar.VarADR),SIZEOF(Internal.ParElement[Internal.i].GenVar.VarADR));
				END_CASE;
			END_IF;
		END_FOR;
		brsmemcpy(Internal.CmdPvAddress,ADR(Internal.Enable),1);
		brsmemcpy(ADR(Internal.Element.Json),pJsonString,SIZEOF(Internal.Element.Json));
		brsmemcpy(pElement,ADR(Internal.Element),SIZEOF(Internal.Element));
	END_IF;
END_FUNCTION
```

#### TC_Seq_Add.st
```iecst
(*  *)
FUNCTION TC_Seq_Add
	//brsmemset(ADR(Internal),0,SIZEOF(Internal));
	TC_Seq_Add := -1;
	IF pJsonArray <> 0 AND pJson <> 0 THEN
		brsmemmove(pJsonArray+DINT_TO_UDINT(MAX_TC_SEQ_JSON_STRING_LEN+1),pJsonArray,DINT_TO_UDINT((MAX_TC_SEQ_JSON_STRING_LEN+1)*MAX_TC_SEQ_BUFFER_IDX));
		brsmemset(pJsonArray,0,DINT_TO_UDINT(MAX_TC_SEQ_JSON_STRING_LEN+1));
		brsmemcpy(pJsonArray,pJson,DINT_TO_UDINT(MAX_TC_SEQ_JSON_STRING_LEN+1));
		TC_Seq_Add := 0;
	END_IF;
END_FUNCTION
```

#### TC_Seq_AddFront.st
```iecst
(*  *)
FUNCTION TC_Seq_AddFront
	brsmemset(ADR(Internal),0,SIZEOF(Internal));
	TC_Seq_AddFront := -1;
	IF pJsonArray <> 0 AND pJson <> 0 THEN
		IF brsstrlen(pJson) > 0 THEN
			FOR Internal.i := MAX_TC_SEQ_BUFFER_IDX TO 0 BY -1 DO
				IF brsstrlen(pJsonArray+DINT_TO_UDINT(Internal.i*(MAX_TC_SEQ_JSON_STRING_LEN+1))) > 0 THEN
					brsmemset(pJsonArray+DINT_TO_UDINT((MAX_TC_SEQ_JSON_STRING_LEN+1)*Internal.i),0,DINT_TO_UDINT(MAX_TC_SEQ_JSON_STRING_LEN+1));
					brsmemcpy(pJsonArray+DINT_TO_UDINT((MAX_TC_SEQ_JSON_STRING_LEN+1)*Internal.i),pJson,DINT_TO_UDINT(MAX_TC_SEQ_JSON_STRING_LEN+1));
					TC_Seq_AddFront := 0;
				END_IF;
			END_FOR;
		END_IF
	END_IF;
END_FUNCTION
```

### Library Logical/Libraries/TC_RAND (ANSIC, version 1.0.0)

#### SRAND.c
```c
#include <bur/plctypes.h>
#include <stdlib.h>
#ifdef __cplusplus
	extern "C"
	{
#endif
	#include "TC_RAND.h"
#ifdef __cplusplus
	};
#endif
/* seed function */
plcbit SRAND(unsigned short Seed)
{
	srand(Seed);
	return 1;
}
```

#### RAND.c
```c
#include <bur/plctypes.h>
#include <stdlib.h>
#ifdef __cplusplus
	extern "C"
	{
#endif
	#include "TC_RAND.h"
#ifdef __cplusplus
	};
#endif
/* Generates random number */
signed short RAND(void)
{
	return (signed short)rand();
}
```

#### RRAND.c
```c
#include <bur/plctypes.h>
#include <stdlib.h>
#ifdef __cplusplus
	extern "C"
	{
#endif
	#include "TC_RAND.h"
#ifdef __cplusplus
	};
#endif
/* Generates random number between the (low,high) */
double RRAND(double low, double high)
{
	return (((double)rand())/2147483647.0)*(high-low)+low;
}
```

#### DRAND.c
```c
#include <bur/plctypes.h>
#include <stdlib.h>
#ifdef __cplusplus
	extern "C"
	{
#endif
	#include "TC_RAND.h"
#ifdef __cplusplus
	};
#endif
/* Generates random number between the (low,high) */
signed long DRAND(signed long low, signed long high)
{
	return (rand() % (high - low + 1)) + low;
}
```

### Library Logical/Libraries/HA_Matrix (IEC)
Depends on: AsBrStr

#### Types.typ - Exported data types
```iecst
TYPE
	HA_Matrix_Array_typ : 	STRUCT
		M : ARRAY[0..MAX_HA_MATRIX_ARRAY_IDX]OF LREAL;
		Row : DINT;
		Col : DINT;
	END_STRUCT;
	HA_Matrix_Internal_typ : 	STRUCT
		sizeArray : UDINT;
		sizeTotal : UDINT;
		row1 : DINT;
		row2 : DINT;
		row3 : DINT;
		row4 : DINT;
		col1 : DINT;
		col2 : DINT;
		col3 : DINT;
		col4 : DINT;
		i1 : DINT;
		i2 : DINT;
		i3 : DINT;
		i4 : DINT;
		temp1 : LREAL;
		temp2 : LREAL;
		temp3 : LREAL;
		temp4 : LREAL;
		temp5 : LREAL;
		result : LREAL;
	END_STRUCT;
	NGRC_Config_typ : 	STRUCT
		LagOrder : DINT := 2;
		PolyOrder : DINT := 2;
		Stride : DINT := 1;
		Lambda : LREAL := 2.5E-6;
		UseBias : BOOL := TRUE;
		UseDerivative : BOOL := TRUE;
		WarmupSteps : DINT := 0;
	END_STRUCT;
	NGRC_Status_enum :
		(
		NGRC_IDLE := 0,
		NGRC_TRAINING := 1,
		NGRC_TRAINED := 2,
		NGRC_PREDICTING := 3,
		NGRC_ERROR := 99
		);
	NGRC_Error_enum :
		(
		NGRC_ERR_NONE := 0,
		NGRC_ERR_NO_DATA := 1,
		NGRC_ERR_INVALID_CONFIG := 2,
		NGRC_ERR_INSUFFICIENT_DATA := 3,
		NGRC_ERR_TRAINING_FAILED := 4,
		NGRC_ERR_PREDICTION_FAILED := 5,
		NGRC_ERR_NOT_TRAINED := 6,
		NGRC_ERR_MEMORY := 7
		);
	NGRC_Internal_typ : 	STRUCT
		Beta : HA_Matrix_Array_typ;
		XtX : HA_Matrix_Array_typ;
		XtY : HA_Matrix_Array_typ;
		L : HA_Matrix_Array_typ;
		LagWork : HA_Matrix_Array_typ;
		PolyWork : HA_Matrix_Array_typ;
		FeatWork : HA_Matrix_Array_typ;
		Ywork : HA_Matrix_Array_typ;
		PredWork : HA_Matrix_Array_typ;
		State : HA_Matrix_Array_typ;
		History : HA_Matrix_Array_typ;
		WorkState : HA_Matrix_Array_typ;
		WorkHist : HA_Matrix_Array_typ;
		TrainStep : DINT;
	END_STRUCT;
	NGRC_Stats_typ : 	STRUCT
		TrainRMSE : LREAL;
		TrainR2 : LREAL;
		LastPredTime : UDINT;
		LastTrainTime : UDINT;
		NumFeatures : DINT;
		NumSamples : DINT;
	END_STRUCT;
	NGRC_Continuous_Config_typ : 	STRUCT
		TrainingSamples : DINT := 200;
		BufferSize : DINT := 500;
		RetrainMode : DINT := 1;
		RetrainInterval : DINT := 50;
		RetrainErrorThreshold : LREAL := 0.1;
		PredictSteps : DINT := 5;
		MultiStepUpdateInterval : DINT := 5;
		ModelConfig : NGRC_Config_typ;
	END_STRUCT;
	NGRC_Continuous_Metrics_typ : 	STRUCT
		OneStepRMSE : LREAL;
		OneStepMaxError : LREAL;
		FiveStepRMSE : LREAL;
		MovingAvgError : LREAL;
		StepErrors : ARRAY[0..4]OF LREAL;
		SampleCount : DINT;
		TotalRetrains : DINT;
		ModelSwaps : DINT;
		TrainingCycles : DINT;
	END_STRUCT;
	NGRC_Continuous_Status_typ : 	STRUCT
		Ready : BOOL;
		PredictionValid : BOOL;
		IsTraining : BOOL;
		TrainingProgress : DINT;
		LastRetrainReason : STRING[40];
	END_STRUCT;
	StateFlags_typ : STRUCT
		Initialized : BOOL := FALSE;
		ActiveModelValid : BOOL := FALSE;
		PredictionActive : BOOL := FALSE;
	END_STRUCT;
	NGRC_MultiVar_Config_typ : STRUCT
		NumVariables : DINT := 1;
		MaxVariables : DINT := 10;
		TrainingSamples : DINT := 200;
		BufferSize : DINT := 500;
		RetrainMode : DINT := 1;
		RetrainInterval : DINT := 50;
		RetrainErrorThreshold : REAL := 0.1;
		PredictSteps : DINT := 5;
		MultiStepUpdateInterval : DINT := 5;
		ModelConfig : NGRC_Config_typ;
	END_STRUCT;
	NGRC_MultiVar_Metrics_typ : STRUCT
		OneStepRMSE : ARRAY[0..9] OF LREAL;
		OneStepMaxError : ARRAY[0..9] OF LREAL;
		FiveStepRMSE : ARRAY[0..9] OF LREAL;
		OverallRMSE : LREAL;
		MovingAvgError : LREAL;
		StepErrors : ARRAY[0..9, 0..4] OF LREAL;
		SampleCount : DINT;
		TotalRetrains : DINT;
		ModelSwaps : DINT;
		TrainingCycles : DINT;
	END_STRUCT;
	NGRC_MultiVar_Status_typ : STRUCT
		Ready : BOOL;
		PredictionValid : BOOL;
		IsTraining : BOOL;
		TrainingProgress : DINT;
		LastRetrainReason : STRING[40];
		ConfigValid : BOOL;
	END_STRUCT;
END_TYPE
```

#### Constants.var - Exported constants
```iecst
VAR CONSTANT
	MAX_HA_MATRIX_ARRAY_IDX : UDINT := 5999;
END_VAR
```
